LIN {X 0,Y 305.411,Z 367.044,A -85,B 0,C 180,E1 -16061.862,E2 -16061.862} C_VEL
LIN {X 0,Y 305.412,Z 367.294,A -85,B 0,C 180,E1 -16065.224,E2 -16065.224} C_VEL
LIN {X 0,Y 309.317,Z 377.708,A -85,B 0,C 180,E1 -16068.083,E2 -16068.083} C_VEL
LIN {X 0,Y 313.501,Z 390,A -85,B 0,C 180,E1 -16071.119,E2 -16071.119} C_VEL
LIN {X 0,Y 315.442,Z 396.314,A -85,B 0,C 180,E1 -16072.486,E2 -16072.486} C_VEL
LIN {X 0,Y 323.182,Z 411.941,A -85,B 0,C 180,E1 -16073.957,E2 -16073.957} C_VEL
LIN {X 0,Y 328.092,Z 423.496,A -85,B 0,C 180,E1 -16074.88,E2 -16074.88} C_VEL
LIN {X 0,Y 331.537,Z 444.039,A -85,B 0,C 180,E1 -16075.825,E2 -16075.825} C_VEL
LIN {X 0,Y 328.819,Z 524.988,A -85,B 0,C 180,E1 -16077.585,E2 -16077.585} C_VEL
LIN {X 0,Y 327.29,Z 565.254,A -85,B 0,C 180,E1 -16078.483,E2 -16078.483} C_VEL
LIN {X 0,Y 326.153,Z 580.481,A -85,B 0,C 180,E1 -16079.038,E2 -16079.038} C_VEL
LIN {X 0,Y 324.598,Z 594.646,A -85,B 0,C 180,E1 -16079.775,E2 -16079.775} C_VEL
LIN {X 0,Y 322.707,Z 608.869,A -85,B 0,C 180,E1 -16080.766,E2 -16080.766} C_VEL
LIN {X 0,Y 320.772,Z 621.593,A -85,B 0,C 180,E1 -16081.897,E2 -16081.897} C_VEL
LIN {X 0,Y 318.404,Z 634.299,A -85,B 0,C 180,E1 -16083.273,E2 -16083.273} C_VEL
LIN {X 0,Y 315.823,Z 647.117,A -85,B 0,C 180,E1 -16084.988,E2 -16084.988} C_VEL
LIN {X 0,Y 313.322,Z 658.678,A -85,B 0,C 180,E1 -16086.876,E2 -16086.876} C_VEL
LIN {X 0,Y 311.244,Z 668.516,A -85,B 0,C 180,E1 -16088.821,E2 -16088.821} C_VEL
LIN {X 0,Y 309.016,Z 678.081,A -85,B 0,C 180,E1 -16091.089,E2 -16091.089} C_VEL
LIN {X 0,Y 307.253,Z 686.052,A -85,B 0,C 180,E1 -16093.386,E2 -16093.386} C_VEL
LIN {X 0,Y 305.786,Z 693.474,A -85,B 0,C 180,E1 -16096.035,E2 -16096.035} C_VEL
LIN {X 0,Y 304.663,Z 699.365,A -85,B 0,C 180,E1 -16098.692,E2 -16098.692} C_VEL
LIN {X 0,Y 304.167,Z 702.846,A -85,B 0,C 180,E1 -16100.692,E2 -16100.692} C_VEL
LIN {X 0,Y 303.722,Z 706.396,A -85,B 0,C 180,E1 -16103.356,E2 -16103.356} C_VEL
LIN {X 0,Y 303.569,Z 708.739,A -85,B 0,C 180,E1 -16106.017,E2 -16106.017} C_VEL
LIN {X 0,Y 303.524,Z 709.928,A -85,B 0,C 180,E1 -16108.673,E2 -16108.673} C_VEL
LIN {X 0,Y 303.524,Z 709.94,A -85,B 0,C 180,E1 -16111.327,E2 -16111.327} C_VEL
LIN {X 0,Y 303.573,Z 708.8,A -85,B 0,C 180,E1 -16113.982,E2 -16113.982} C_VEL
LIN {X 0,Y 303.725,Z 706.51,A -85,B 0,C 180,E1 -16116.644,E2 -16116.644} C_VEL
LIN {X 0,Y 304.16,Z 703.02,A -85,B 0,C 180,E1 -16119.308,E2 -16119.308} C_VEL
LIN {X 0,Y 304.837,Z 698.241,A -85,B 0,C 180,E1 -16121.975,E2 -16121.975} C_VEL
LIN {X 0,Y 306.042,Z 692.044,A -85,B 0,C 180,E1 -16124.632,E2 -16124.632} C_VEL
LIN {X 0,Y 307.409,Z 685.357,A -85,B 0,C 180,E1 -16126.947,E2 -16126.947} C_VEL
LIN {X 0,Y 309.208,Z 677.258,A -85,B 0,C 180,E1 -16129.243,E2 -16129.243} C_VEL
LIN {X 0,Y 311.526,Z 667.524,A -85,B 0,C 180,E1 -16131.506,E2 -16131.506} C_VEL
LIN {X 0,Y 313.768,Z 656.8,A -85,B 0,C 180,E1 -16133.576,E2 -16133.576} C_VEL
LIN {X 0,Y 316.463,Z 644.635,A -85,B 0,C 180,E1 -16135.485,E2 -16135.485} C_VEL
LIN {X 0,Y 319.039,Z 631.238,A -85,B 0,C 180,E1 -16137.2,E2 -16137.2} C_VEL
LIN {X 0,Y 319.416,Z 629.216,A -85,B 0,C 180,E1 -16137.422,E2 -16137.422} C_VEL
LIN {X 0,Y 319.706,Z 624.316,A -85,B 0,C 180,E1 -16138.005,E2 -16138.005} C_VEL
LIN {X 0,Y 318.605,Z 616.252,A -85,B 0,C 180,E1 -16139.03,E2 -16139.03} C_VEL
LIN {X 0,Y 317.409,Z 607.963,A -85,B 0,C 180,E1 -16139.981,E2 -16139.981} C_VEL
LIN {X 0,Y 317.523,Z 602.64,A -85,B 0,C 180,E1 -16140.441,E2 -16140.441} C_VEL
LIN {X 0,Y 319.252,Z 588.464,A -85,B 0,C 180,E1 -16141.338,E2 -16141.338} C_VEL
LIN {X 0,Y 320.747,Z 573.705,A -85,B 0,C 180,E1 -16142.004,E2 -16142.004} C_VEL
LIN {X 0,Y 321.69,Z 558.805,A -85,B 0,C 180,E1 -16142.454,E2 -16142.454} C_VEL
LIN {X 0,Y 325.778,Z 445.6,A -85,B 0,C 180,E1 -16144.938,E2 -16144.938} C_VEL
LIN {X 0,Y 322.373,Z 425.482,A -85,B 0,C 180,E1 -16145.9,E2 -16145.9} C_VEL
LIN {X 0,Y 315.354,Z 409.904,A -85,B 0,C 180,E1 -16147.259,E2 -16147.259} C_VEL
LIN {X 0,Y 308.177,Z 395.852,A -85,B 0,C 180,E1 -16148.71,E2 -16148.71} C_VEL
LIN {X 0,Y 304.501,Z 384.759,A -85,B 0,C 180,E1 -16151.401,E2 -16151.401} C_VEL
LIN {X 0,Y 300.748,Z 374.308,A -85,B 0,C 180,E1 -16154.188,E2 -16154.188} C_VEL
LIN {X 0,Y 298.408,Z 368.151,A -85,B 0,C 180,E1 -16155.992,E2 -16155.992} C_VEL
LIN {X 0,Y 298.348,Z 367.948,A -85,B 0,C 180,E1 -16158.921,E2 -16158.921} C_VEL
LIN {X 0,Y 298.386,Z 367.941,A -85,B 0,C 180,E1 -16162.237,E2 -16162.237} C_VEL
LIN {X 0,Y 298.407,Z 367.933,A -85,B 0,C 180,E1 -16165.581,E2 -16165.581} C_VEL
LIN {X 0,Y 298.376,Z 367.928,A -85,B 0,C 180,E1 -16168.789,E2 -16168.789} C_VEL
LIN {X 0,Y 298.413,Z 367.926,A -85,B 0,C 180,E1 -16171.899,E2 -16171.899} C_VEL
LIN {X 0,Y 298.439,Z 367.934,A -85,B 0,C 180,E1 -16174.92,E2 -16174.92} C_VEL
LIN {X 0,Y 298.401,Z 367.92,A -85,B 0,C 180,E1 -16177.862,E2 -16177.862} C_VEL
LIN {X 0,Y 298.503,Z 367.927,A -85,B 0,C 180,E1 -16180.754,E2 -16180.754} C_VEL
LIN {X 0,Y 298.586,Z 367.911,A -85,B 0,C 180,E1 -16184.994,E2 -16184.994} C_VEL
LIN {X 0,Y 298.583,Z 367.892,A -85,B 0,C 180,E1 -16189.146,E2 -16189.146} C_VEL
LIN {X 0,Y 298.719,Z 367.902,A -85,B 0,C 180,E1 -16191.885,E2 -16191.885} C_VEL
LIN {X 0,Y 298.648,Z 367.885,A -85,B 0,C 180,E1 -16194.599,E2 -16194.599} C_VEL
LIN {X 0,Y 298.92,Z 367.875,A -85,B 0,C 180,E1 -16198.653,E2 -16198.653} C_VEL
LIN {X 0,Y 298.921,Z 367.849,A -85,B 0,C 180,E1 -16201.347,E2 -16201.347} C_VEL
LIN {X 0,Y 298.641,Z 367.905,A -85,B 0,C 180,E1 -16205.401,E2 -16205.401} C_VEL
LIN {X 0,Y 298.702,Z 367.875,A -85,B 0,C 180,E1 -16208.115,E2 -16208.115} C_VEL
LIN {X 0,Y 298.551,Z 367.909,A -85,B 0,C 180,E1 -16212.231,E2 -16212.231} C_VEL
LIN {X 0,Y 298.55,Z 367.905,A -85,B 0,C 180,E1 -16215.169,E2 -16215.169} C_VEL
LIN {X 0,Y 298.504,Z 367.905,A -85,B 0,C 180,E1 -16219.245,E2 -16219.245} C_VEL
LIN {X 0,Y 298.458,Z 367.924,A -85,B 0,C 180,E1 -16223.597,E2 -16223.597} C_VEL
LIN {X 0,Y 298.489,Z 367.924,A -85,B 0,C 180,E1 -16226.574,E2 -16226.574} C_VEL
LIN {X 0,Y 298.42,Z 367.92,A -85,B 0,C 180,E1 -16229.641,E2 -16229.641} C_VEL
LIN {X 0,Y 298.395,Z 367.939,A -85,B 0,C 180,E1 -16232.8,E2 -16232.8} C_VEL
LIN {X 0,Y 298.444,Z 367.935,A -85,B 0,C 180,E1 -16236.807,E2 -16236.807} C_VEL
LIN {X 0,Y 298.386,Z 367.89,A -85,B 0,C 180,E1 -16241.088,E2 -16241.088} C_VEL
LIN {X 0,Y 298.398,Z 367.931,A -85,B 0,C 180,E1 -16243.103,E2 -16243.103} C_VEL
LIN {X 0,Y 298.432,Z 368.054,A -85,B 0,C 180,E1 -16247.297,E2 -16247.297} C_VEL
LIN {X 0,Y 298.626,Z 368.899,A -85,B 0,C 180,E1 -16247.593,E2 -16247.593} C_VEL
LIN {X 0,Y 302.505,Z 376.069,A -85,B 0,C 180,E1 -16249.032,E2 -16249.032} C_VEL
LIN {X 0,Y 308.412,Z 392.412,A -85,B 0,C 180,E1 -16251.566,E2 -16251.566} C_VEL
LIN {X 0,Y 316.344,Z 409.427,A -85,B 0,C 180,E1 -16253.177,E2 -16253.177} C_VEL
LIN {X 0,Y 322.801,Z 424.458,A -85,B 0,C 180,E1 -16254.439,E2 -16254.439} C_VEL
LIN {X 0,Y 325.22,Z 441.813,A -85,B 0,C 180,E1 -16255.203,E2 -16255.203} C_VEL
LIN {X 0,Y 320.9,Z 562.756,A -85,B 0,C 180,E1 -16257.874,E2 -16257.874} C_VEL
LIN {X 0,Y 319.802,Z 578.013,A -85,B 0,C 180,E1 -16258.4,E2 -16258.4} C_VEL
LIN {X 0,Y 318.3,Z 592.161,A -85,B 0,C 180,E1 -16259.113,E2 -16259.113} C_VEL
LIN {X 0,Y 316.442,Z 606.126,A -85,B 0,C 180,E1 -16260.06,E2 -16260.06} C_VEL
LIN {X 0,Y 314.307,Z 619.886,A -85,B 0,C 180,E1 -16261.266,E2 -16261.266} C_VEL
LIN {X 0,Y 311.853,Z 632.809,A -85,B 0,C 180,E1 -16262.666,E2 -16262.666} C_VEL
LIN {X 0,Y 309.452,Z 644.715,A -85,B 0,C 180,E1 -16264.256,E2 -16264.256} C_VEL
LIN {X 0,Y 307.017,Z 655.77,A -85,B 0,C 180,E1 -16266.037,E2 -16266.037} C_VEL
LIN {X 0,Y 304.805,Z 665.842,A -85,B 0,C 180,E1 -16267.995,E2 -16267.995} C_VEL
LIN {X 0,Y 302.413,Z 675.711,A -85,B 0,C 180,E1 -16270.307,E2 -16270.307} C_VEL
LIN {X 0,Y 300.504,Z 683.894,A -85,B 0,C 180,E1 -16272.651,E2 -16272.651} C_VEL
LIN {X 0,Y 299.073,Z 690.659,A -85,B 0,C 180,E1 -16275.02,E2 -16275.02} C_VEL
LIN {X 0,Y 297.826,Z 696.924,A -85,B 0,C 180,E1 -16277.738,E2 -16277.738} C_VEL
LIN {X 0,Y 297.095,Z 701.755,A -85,B 0,C 180,E1 -16280.469,E2 -16280.469} C_VEL
LIN {X 0,Y 296.647,Z 705.286,A -85,B 0,C 180,E1 -16283.197,E2 -16283.197} C_VEL
LIN {X 0,Y 296.482,Z 707.609,A -85,B 0,C 180,E1 -16285.922,E2 -16285.922} C_VEL
LIN {X 0,Y 296.458,Z 708.776,A -85,B 0,C 180,E1 -16288.642,E2 -16288.642} C_VEL
LIN {X 0,Y 296.458,Z 708.774,A -85,B 0,C 180,E1 -16291.359,E2 -16291.359} C_VEL
LIN {X 0,Y 296.483,Z 707.601,A -85,B 0,C 180,E1 -16294.078,E2 -16294.078} C_VEL
LIN {X 0,Y 296.647,Z 705.268,A -85,B 0,C 180,E1 -16296.803,E2 -16296.803} C_VEL
LIN {X 0,Y 297.095,Z 701.72,A -85,B 0,C 180,E1 -16299.532,E2 -16299.532} C_VEL
LIN {X 0,Y 297.834,Z 696.875,A -85,B 0,C 180,E1 -16302.262,E2 -16302.262} C_VEL
LIN {X 0,Y 299.073,Z 690.605,A -85,B 0,C 180,E1 -16304.981,E2 -16304.981} C_VEL
LIN {X 0,Y 300.794,Z 682.716,A -85,B 0,C 180,E1 -16307.683,E2 -16307.683} C_VEL
LIN {X 0,Y 302.715,Z 674.287,A -85,B 0,C 180,E1 -16310.026,E2 -16310.026} C_VEL
LIN {X 0,Y 308.167,Z 654.094,A -85,B 0,C 180,E1 -16314.596,E2 -16314.596} C_VEL
LIN {X 0,Y 311.872,Z 642.327,A -85,B 0,C 180,E1 -16316.789,E2 -16316.789} C_VEL
LIN {X 0,Y 315.458,Z 630.417,A -85,B 0,C 180,E1 -16318.62,E2 -16318.62} C_VEL
LIN {X 0,Y 319.129,Z 617.583,A -85,B 0,C 180,E1 -16320.25,E2 -16320.25} C_VEL
LIN {X 0,Y 322.798,Z 603.816,A -85,B 0,C 180,E1 -16321.678,E2 -16321.678} C_VEL
LIN {X 0,Y 326.682,Z 587.895,A -85,B 0,C 180,E1 -16322.987,E2 -16322.987} C_VEL
LIN {X 0,Y 330.115,Z 572.099,A -85,B 0,C 180,E1 -16323.977,E2 -16323.977} C_VEL
LIN {X 0,Y 332.855,Z 556.74,A -85,B 0,C 180,E1 -16324.71,E2 -16324.71} C_VEL
LIN {X 0,Y 342.563,Z 489.987,A -85,B 0,C 180,E1 -16327.245,E2 -16327.245} C_VEL
LIN {X 0,Y 348.996,Z 451.001,A -85,B 0,C 180,E1 -16328.721,E2 -16328.721} C_VEL
LIN {X 0,Y 347.231,Z 446.356,A -85,B 0,C 180,E1 -16330.058,E2 -16330.058} C_VEL
LIN {X 0,Y 345.905,Z 443.202,A -85,B 0,C 180,E1 -16331.257,E2 -16331.257} C_VEL
LIN {X 0,Y 344.191,Z 439.714,A -85,B 0,C 180,E1 -16333.319,E2 -16333.319} C_VEL
LIN {X 0,Y 343.35,Z 438.48,A -85,B 0,C 180,E1 -16335.002,E2 -16335.002} C_VEL
LIN {X 0,Y 343.223,Z 438.552,A -85,B 0,C 180,E1 -16337.49,E2 -16337.49} C_VEL
LIN {X 0,Y 343.926,Z 439.872,A -85,B 0,C 180,E1 -16339.267,E2 -16339.267} C_VEL
LIN {X 0,Y 345.698,Z 444.259,A -85,B 0,C 180,E1 -16341.637,E2 -16341.637} C_VEL
LIN {X 0,Y 347.324,Z 448.856,A -85,B 0,C 180,E1 -16343.179,E2 -16343.179} C_VEL
LIN {X 0,Y 348.467,Z 452.55,A -85,B 0,C 180,E1 -16344.127,E2 -16344.127} C_VEL
LIN {X 0,Y 348.241,Z 454.474,A -85,B 0,C 180,E1 -16344.255,E2 -16344.255} C_VEL
LIN {X 0,Y 334.114,Z 539.694,A -85,B 0,C 180,E1 -16347.718,E2 -16347.718} C_VEL
LIN {X 0,Y 331.471,Z 555.843,A -85,B 0,C 180,E1 -16348.469,E2 -16348.469} C_VEL
LIN {X 0,Y 328.38,Z 571.369,A -85,B 0,C 180,E1 -16349.45,E2 -16349.45} C_VEL
LIN {X 0,Y 324.96,Z 586.557,A -85,B 0,C 180,E1 -16350.704,E2 -16350.704} C_VEL
LIN {X 0,Y 321.371,Z 600.391,A -85,B 0,C 180,E1 -16352.132,E2 -16352.132} C_VEL
LIN {X 0,Y 317.77,Z 613.05,A -85,B 0,C 180,E1 -16353.747,E2 -16353.747} C_VEL
LIN {X 0,Y 314.257,Z 624.641,A -85,B 0,C 180,E1 -16355.561,E2 -16355.561} C_VEL
LIN {X 0,Y 311.147,Z 634.413,A -85,B 0,C 180,E1 -16357.419,E2 -16357.419} C_VEL
LIN {X 0,Y 307.886,Z 644.112,A -85,B 0,C 180,E1 -16359.659,E2 -16359.659} C_VEL
LIN {X 0,Y 305.091,Z 651.899,A -85,B 0,C 180,E1 -16361.882,E2 -16361.882} C_VEL
LIN {X 0,Y 302.424,Z 659.117,A -85,B 0,C 180,E1 -16364.5,E2 -16364.5} C_VEL
LIN {X 0,Y 300.431,Z 664.653,A -85,B 0,C 180,E1 -16367.16,E2 -16367.16} C_VEL
LIN {X 0,Y 299.358,Z 667.8,A -85,B 0,C 180,E1 -16369.175,E2 -16369.175} C_VEL
LIN {X 0,Y 298.079,Z 670.711,A -85,B 0,C 180,E1 -16371.867,E2 -16371.867} C_VEL
LIN {X 0,Y 297.263,Z 672.207,A -85,B 0,C 180,E1 -16374.574,E2 -16374.574} C_VEL
LIN {X 0,Y 296.912,Z 672.286,A -85,B 0,C 180,E1 -16377.287,E2 -16377.287} C_VEL
LIN {X 0,Y 296.668,Z 670.948,A -85,B 0,C 180,E1 -16380,E2 -16380} C_VEL
LIN {X 0,Y 296.698,Z 668.154,A -85,B 0,C 180,E1 -16382.716,E2 -16382.716} C_VEL
LIN {X 0,Y 296.784,Z 665.05,A -85,B 0,C 180,E1 -16384.754,E2 -16384.754} C_VEL
LIN {X 0,Y 297.063,Z 660.107,A -85,B 0,C 180,E1 -16387.199,E2 -16387.199} C_VEL
LIN {X 0,Y 297.439,Z 654.084,A -85,B 0,C 180,E1 -16389.521,E2 -16389.521} C_VEL
LIN {X 0,Y 298.097,Z 646.353,A -85,B 0,C 180,E1 -16391.905,E2 -16391.905} C_VEL
LIN {X 0,Y 299.015,Z 638.312,A -85,B 0,C 180,E1 -16393.941,E2 -16393.941} C_VEL
LIN {X 0,Y 299.934,Z 628.773,A -85,B 0,C 180,E1 -16395.956,E2 -16395.956} C_VEL
LIN {X 0,Y 301.307,Z 617.06,A -85,B 0,C 180,E1 -16398.003,E2 -16398.003} C_VEL
LIN {X 0,Y 302.519,Z 605.387,A -85,B 0,C 180,E1 -16399.686,E2 -16399.686} C_VEL
LIN {X 0,Y 303.938,Z 592.777,A -85,B 0,C 180,E1 -16401.18,E2 -16401.18} C_VEL
LIN {X 0,Y 305.32,Z 579.078,A -85,B 0,C 180,E1 -16402.5,E2 -16402.5} C_VEL
LIN {X 0,Y 306.468,Z 564.482,A -85,B 0,C 180,E1 -16403.618,E2 -16403.618} C_VEL
LIN {X 0,Y 307.548,Z 548.938,A -85,B 0,C 180,E1 -16404.513,E2 -16404.513} C_VEL
LIN {X 0,Y 308.473,Z 531.327,A -85,B 0,C 180,E1 -16405.199,E2 -16405.199} C_VEL
LIN {X 0,Y 313.035,Z 438.431,A -85,B 0,C 180,E1 -16408.326,E2 -16408.326} C_VEL
LIN {X 0,Y 308.171,Z 405.676,A -85,B 0,C 180,E1 -16409.875,E2 -16409.875} C_VEL
LIN {X 0,Y 305.512,Z 398.037,A -85,B 0,C 180,E1 -16410.404,E2 -16410.404} C_VEL
LIN {X 0,Y 302.475,Z 384.617,A -85,B 0,C 180,E1 -16413.893,E2 -16413.893} C_VEL
LIN {X 0,Y 299.638,Z 372.911,A -85,B 0,C 180,E1 -16417.111,E2 -16417.111} C_VEL
LIN {X 0,Y 298.443,Z 368.214,A -85,B 0,C 180,E1 -16418.494,E2 -16418.494} C_VEL
LIN {X 0,Y 298.375,Z 367.944,A -85,B 0,C 180,E1 -16419.492,E2 -16419.492} C_VEL
LIN {X 0,Y 298.371,Z 367.944,A -85,B 0,C 180,E1 -16423.781,E2 -16423.781} C_VEL
LIN {X 0,Y 298.435,Z 368.42,A -85,B 0,C 180,E1 -16424.239,E2 -16424.239} C_VEL
LIN {X 0,Y 302.771,Z 379.718,A -85,B 0,C 180,E1 -16427.427,E2 -16427.427} C_VEL
LIN {X 0,Y 307.254,Z 392.856,A -85,B 0,C 180,E1 -16430.733,E2 -16430.733} C_VEL
LIN {X 0,Y 308.293,Z 396.188,A -85,B 0,C 180,E1 -16431.459,E2 -16431.459} C_VEL
LIN {X 0,Y 316.348,Z 411.985,A -85,B 0,C 180,E1 -16433.056,E2 -16433.056} C_VEL
LIN {X 0,Y 322.396,Z 425.621,A -85,B 0,C 180,E1 -16434.225,E2 -16434.225} C_VEL
LIN {X 0,Y 325.662,Z 445.137,A -85,B 0,C 180,E1 -16435.152,E2 -16435.152} C_VEL
LIN {X 0,Y 322.86,Z 525.012,A -85,B 0,C 180,E1 -16436.914,E2 -16436.914} C_VEL
LIN {X 0,Y 321.263,Z 565.177,A -85,B 0,C 180,E1 -16437.822,E2 -16437.822} C_VEL
LIN {X 0,Y 320.096,Z 580.432,A -85,B 0,C 180,E1 -16438.385,E2 -16438.385} C_VEL
LIN {X 0,Y 318.479,Z 594.609,A -85,B 0,C 180,E1 -16439.131,E2 -16439.131} C_VEL
LIN {X 0,Y 316.442,Z 609.431,A -85,B 0,C 180,E1 -16440.185,E2 -16440.185} C_VEL
LIN {X 0,Y 314.24,Z 623.112,A -85,B 0,C 180,E1 -16441.441,E2 -16441.441} C_VEL
LIN {X 0,Y 311.789,Z 635.543,A -85,B 0,C 180,E1 -16442.841,E2 -16442.841} C_VEL
LIN {X 0,Y 309.137,Z 648.15,A -85,B 0,C 180,E1 -16444.589,E2 -16444.589} C_VEL
LIN {X 0,Y 306.584,Z 659.378,A -85,B 0,C 180,E1 -16446.483,E2 -16446.483} C_VEL
LIN {X 0,Y 304.59,Z 668.5,A -85,B 0,C 180,E1 -16448.335,E2 -16448.335} C_VEL
LIN {X 0,Y 302.248,Z 678.066,A -85,B 0,C 180,E1 -16450.649,E2 -16450.649} C_VEL
LIN {X 0,Y 300.369,Z 686.037,A -85,B 0,C 180,E1 -16452.994,E2 -16452.994} C_VEL
LIN {X 0,Y 298.835,Z 693.46,A -85,B 0,C 180,E1 -16455.703,E2 -16455.703} C_VEL
LIN {X 0,Y 297.64,Z 699.351,A -85,B 0,C 180,E1 -16458.422,E2 -16458.422} C_VEL
LIN {X 0,Y 297.108,Z 702.832,A -85,B 0,C 180,E1 -16460.469,E2 -16460.469} C_VEL
LIN {X 0,Y 296.646,Z 706.383,A -85,B 0,C 180,E1 -16463.197,E2 -16463.197} C_VEL
LIN {X 0,Y 296.471,Z 708.725,A -85,B 0,C 180,E1 -16465.922,E2 -16465.922} C_VEL
LIN {X 0,Y 296.446,Z 709.914,A -85,B 0,C 180,E1 -16468.641,E2 -16468.641} C_VEL
LIN {X 0,Y 296.446,Z 709.926,A -85,B 0,C 180,E1 -16471.358,E2 -16471.358} C_VEL
LIN {X 0,Y 296.476,Z 708.786,A -85,B 0,C 180,E1 -16474.078,E2 -16474.078} C_VEL
LIN {X 0,Y 296.649,Z 706.495,A -85,B 0,C 180,E1 -16476.803,E2 -16476.803} C_VEL
LIN {X 0,Y 297.099,Z 703.005,A -85,B 0,C 180,E1 -16479.531,E2 -16479.531} C_VEL
LIN {X 0,Y 297.856,Z 698.225,A -85,B 0,C 180,E1 -16482.26,E2 -16482.26} C_VEL
LIN {X 0,Y 299.134,Z 692.027,A -85,B 0,C 180,E1 -16484.977,E2 -16484.977} C_VEL
LIN {X 0,Y 300.823,Z 684.238,A -85,B 0,C 180,E1 -16487.681,E2 -16487.681} C_VEL
LIN {X 0,Y 302.774,Z 675.935,A -85,B 0,C 180,E1 -16490.022,E2 -16490.022} C_VEL
LIN {X 0,Y 304.887,Z 667.503,A -85,B 0,C 180,E1 -16491.998,E2 -16491.998} C_VEL
LIN {X 0,Y 307.061,Z 657.467,A -85,B 0,C 180,E1 -16493.982,E2 -16493.982} C_VEL
LIN {X 0,Y 309.793,Z 645.673,A -85,B 0,C 180,E1 -16495.894,E2 -16495.894} C_VEL
LIN {X 0,Y 312.457,Z 632.555,A -85,B 0,C 180,E1 -16497.64,E2 -16497.64} C_VEL
LIN {X 0,Y 314.911,Z 619.45,A -85,B 0,C 180,E1 -16499.039,E2 -16499.039} C_VEL
LIN {X 0,Y 317.19,Z 605.239,A -85,B 0,C 180,E1 -16500.251,E2 -16500.251} C_VEL
LIN {X 0,Y 317.523,Z 602.64,A -85,B 0,C 180,E1 -16500.441,E2 -16500.441} C_VEL
LIN {X 0,Y 317.631,Z 597.225,A -85,B 0,C 180,E1 -16500.883,E2 -16500.883} C_VEL
LIN {X 0,Y 314.9,Z 581.34,A -85,B 0,C 180,E1 -16502.278,E2 -16502.278} C_VEL
LIN {X 0,Y 314.61,Z 575.744,A -85,B 0,C 180,E1 -16502.607,E2 -16502.607} C_VEL
LIN {X 0,Y 314.731,Z 573.829,A -85,B 0,C 180,E1 -16502.682,E2 -16502.682} C_VEL
LIN {X 0,Y 315.719,Z 558.663,A -85,B 0,C 180,E1 -16503.145,E2 -16503.145} C_VEL
LIN {X 0,Y 319.949,Z 446.756,A -85,B 0,C 180,E1 -16505.635,E2 -16505.635} C_VEL
LIN {X 0,Y 316.814,Z 428.216,A -85,B 0,C 180,E1 -16506.551,E2 -16506.551} C_VEL
LIN {X 0,Y 309.707,Z 412.421,A -85,B 0,C 180,E1 -16507.981,E2 -16507.981} C_VEL
LIN {X 0,Y 302.9,Z 399.352,A -85,B 0,C 180,E1 -16509.379,E2 -16509.379} C_VEL
LIN {X 0,Y 300.951,Z 395.526,A -85,B 0,C 180,E1 -16509.851,E2 -16509.851} C_VEL
LIN {X 0,Y 296.548,Z 382.513,A -85,B 0,C 180,E1 -16513.205,E2 -16513.205} C_VEL
LIN {X 0,Y 292.629,Z 372.347,A -85,B 0,C 180,E1 -16516.096,E2 -16516.096} C_VEL
LIN {X 0,Y 291.343,Z 368.975,A -85,B 0,C 180,E1 -16517.189,E2 -16517.189} C_VEL
LIN {X 0,Y 291.332,Z 368.811,A -85,B 0,C 180,E1 -16521.155,E2 -16521.155} C_VEL
LIN {X 0,Y 291.354,Z 368.805,A -85,B 0,C 180,E1 -16524.625,E2 -16524.625} C_VEL
LIN {X 0,Y 291.366,Z 368.802,A -85,B 0,C 180,E1 -16527.95,E2 -16527.95} C_VEL
LIN {X 0,Y 291.345,Z 368.816,A -85,B 0,C 180,E1 -16531.154,E2 -16531.154} C_VEL
LIN {X 0,Y 291.359,Z 368.809,A -85,B 0,C 180,E1 -16534.266,E2 -16534.266} C_VEL
LIN {X 0,Y 291.364,Z 368.797,A -85,B 0,C 180,E1 -16537.298,E2 -16537.298} C_VEL
LIN {X 0,Y 291.44,Z 368.807,A -85,B 0,C 180,E1 -16540.269,E2 -16540.269} C_VEL
LIN {X 0,Y 291.498,Z 368.788,A -85,B 0,C 180,E1 -16544.665,E2 -16544.665} C_VEL
LIN {X 0,Y 291.529,Z 368.77,A -85,B 0,C 180,E1 -16548.88,E2 -16548.88} C_VEL
LIN {X 0,Y 291.668,Z 368.778,A -85,B 0,C 180,E1 -16551.687,E2 -16551.687} C_VEL
LIN {X 0,Y 291.619,Z 368.761,A -85,B 0,C 180,E1 -16554.468,E2 -16554.468} C_VEL
LIN {X 0,Y 291.886,Z 368.751,A -85,B 0,C 180,E1 -16558.62,E2 -16558.62} C_VEL
LIN {X 0,Y 291.887,Z 368.724,A -85,B 0,C 180,E1 -16561.38,E2 -16561.38} C_VEL
LIN {X 0,Y 291.61,Z 368.78,A -85,B 0,C 180,E1 -16565.532,E2 -16565.532} C_VEL
LIN {X 0,Y 291.669,Z 368.757,A -85,B 0,C 180,E1 -16568.912,E2 -16568.912} C_VEL
LIN {X 0,Y 291.517,Z 368.779,A -85,B 0,C 180,E1 -16572.531,E2 -16572.531} C_VEL
LIN {X 0,Y 291.507,Z 368.784,A -85,B 0,C 180,E1 -16575.379,E2 -16575.379} C_VEL
LIN {X 0,Y 291.423,Z 368.786,A -85,B 0,C 180,E1 -16579.86,E2 -16579.86} C_VEL
LIN {X 0,Y 291.4,Z 368.795,A -85,B 0,C 180,E1 -16584.205,E2 -16584.205} C_VEL
LIN {X 0,Y 291.423,Z 368.81,A -85,B 0,C 180,E1 -16587.271,E2 -16587.271} C_VEL
LIN {X 0,Y 291.337,Z 368.803,A -85,B 0,C 180,E1 -16590.437,E2 -16590.437} C_VEL
LIN {X 0,Y 291.344,Z 368.806,A -85,B 0,C 180,E1 -16593.698,E2 -16593.698} C_VEL
LIN {X 0,Y 291.372,Z 368.807,A -85,B 0,C 180,E1 -16597.253,E2 -16597.253} C_VEL
LIN {X 0,Y 291.331,Z 368.764,A -85,B 0,C 180,E1 -16600.643,E2 -16600.643} C_VEL
LIN {X 0,Y 291.29,Z 368.812,A -85,B 0,C 180,E1 -16604.402,E2 -16604.402} C_VEL
LIN {X 0,Y 291.322,Z 368.967,A -85,B 0,C 180,E1 -16606.031,E2 -16606.031} C_VEL
LIN {X 0,Y 291.657,Z 370.251,A -85,B 0,C 180,E1 -16606.428,E2 -16606.428} C_VEL
LIN {X 0,Y 293.268,Z 372.793,A -85,B 0,C 180,E1 -16607.028,E2 -16607.028} C_VEL
LIN {X 0,Y 297.706,Z 381.398,A -85,B 0,C 180,E1 -16608.748,E2 -16608.748} C_VEL
LIN {X 0,Y 301.647,Z 392.41,A -85,B 0,C 180,E1 -16610.533,E2 -16610.533} C_VEL
LIN {X 0,Y 309.608,Z 409.51,A -85,B 0,C 180,E1 -16612.235,E2 -16612.235} C_VEL
LIN {X 0,Y 317.224,Z 426.908,A -85,B 0,C 180,E1 -16613.778,E2 -16613.778} C_VEL
LIN {X 0,Y 319.398,Z 443.039,A -85,B 0,C 180,E1 -16614.502,E2 -16614.502} C_VEL
LIN {X 0,Y 314.925,Z 562.876,A -85,B 0,C 180,E1 -16617.189,E2 -16617.189} C_VEL
LIN {X 0,Y 313.788,Z 578.087,A -85,B 0,C 180,E1 -16617.722,E2 -16617.722} C_VEL
LIN {X 0,Y 312.221,Z 592.215,A -85,B 0,C 180,E1 -16618.443,E2 -16618.443} C_VEL
LIN {X 0,Y 310.35,Z 605.809,A -85,B 0,C 180,E1 -16619.375,E2 -16619.375} C_VEL
LIN {X 0,Y 308.1,Z 619.92,A -85,B 0,C 180,E1 -16620.631,E2 -16620.631} C_VEL
LIN {X 0,Y 305.551,Z 632.838,A -85,B 0,C 180,E1 -16622.054,E2 -16622.054} C_VEL
LIN {X 0,Y 303.046,Z 644.741,A -85,B 0,C 180,E1 -16623.671,E2 -16623.671} C_VEL
LIN {X 0,Y 300.5,Z 655.742,A -85,B 0,C 180,E1 -16625.473,E2 -16625.473} C_VEL
LIN {X 0,Y 298.187,Z 665.863,A -85,B 0,C 180,E1 -16627.481,E2 -16627.481} C_VEL
LIN {X 0,Y 295.7,Z 675.73,A -85,B 0,C 180,E1 -16629.841,E2 -16629.841} C_VEL
LIN {X 0,Y 293.67,Z 683.912,A -85,B 0,C 180,E1 -16632.234,E2 -16632.234} C_VEL
LIN {X 0,Y 292.175,Z 690.676,A -85,B 0,C 180,E1 -16634.657,E2 -16634.657} C_VEL
LIN {X 0,Y 290.858,Z 696.94,A -85,B 0,C 180,E1 -16637.44,E2 -16637.44} C_VEL
LIN {X 0,Y 290.058,Z 701.771,A -85,B 0,C 180,E1 -16640.235,E2 -16640.235} C_VEL
LIN {X 0,Y 289.572,Z 705.301,A -85,B 0,C 180,E1 -16643.03,E2 -16643.03} C_VEL
LIN {X 0,Y 289.388,Z 707.623,A -85,B 0,C 180,E1 -16645.822,E2 -16645.822} C_VEL
LIN {X 0,Y 289.381,Z 708.79,A -85,B 0,C 180,E1 -16648.609,E2 -16648.609} C_VEL
LIN {X 0,Y 289.381,Z 708.788,A -85,B 0,C 180,E1 -16651.392,E2 -16651.392} C_VEL
LIN {X 0,Y 289.389,Z 707.614,A -85,B 0,C 180,E1 -16654.178,E2 -16654.178} C_VEL
LIN {X 0,Y 289.573,Z 705.282,A -85,B 0,C 180,E1 -16656.97,E2 -16656.97} C_VEL
LIN {X 0,Y 290.058,Z 701.734,A -85,B 0,C 180,E1 -16659.765,E2 -16659.765} C_VEL
LIN {X 0,Y 290.867,Z 696.889,A -85,B 0,C 180,E1 -16662.56,E2 -16662.56} C_VEL
LIN {X 0,Y 292.174,Z 690.619,A -85,B 0,C 180,E1 -16665.343,E2 -16665.343} C_VEL
LIN {X 0,Y 293.97,Z 682.731,A -85,B 0,C 180,E1 -16668.107,E2 -16668.107} C_VEL
LIN {X 0,Y 295.972,Z 674.303,A -85,B 0,C 180,E1 -16670.503,E2 -16670.503} C_VEL
LIN {X 0,Y 298.632,Z 664.994,A -85,B 0,C 180,E1 -16672.85,E2 -16672.85} C_VEL
LIN {X 0,Y 301.835,Z 655.393,A -85,B 0,C 180,E1 -16675.147,E2 -16675.147} C_VEL
LIN {X 0,Y 305.718,Z 644.038,A -85,B 0,C 180,E1 -16677.373,E2 -16677.373} C_VEL
LIN {X 0,Y 309.147,Z 633.635,A -85,B 0,C 180,E1 -16679.074,E2 -16679.074} C_VEL
LIN {X 0,Y 313.308,Z 620.392,A -85,B 0,C 180,E1 -16680.872,E2 -16680.872} C_VEL
LIN {X 0,Y 317.523,Z 605.973,A -85,B 0,C 180,E1 -16682.462,E2 -16682.462} C_VEL
LIN {X 0,Y 321.37,Z 591.772,A -85,B 0,C 180,E1 -16683.706,E2 -16683.706} C_VEL
LIN {X 0,Y 325.059,Z 576.525,A -85,B 0,C 180,E1 -16684.743,E2 -16684.743} C_VEL
LIN {X 0,Y 328.185,Z 561.072,A -85,B 0,C 180,E1 -16685.56,E2 -16685.56} C_VEL
LIN {X 0,Y 342.587,Z 472.807,A -85,B 0,C 180,E1 -16688.971,E2 -16688.971} C_VEL
LIN {X 0,Y 345.708,Z 455.092,A -85,B 0,C 180,E1 -16689.677,E2 -16689.677} C_VEL
LIN {X 0,Y 344.22,Z 451.001,A -85,B 0,C 180,E1 -16691.029,E2 -16691.029} C_VEL
LIN {X 0,Y 343.323,Z 448.898,A -85,B 0,C 180,E1 -16691.984,E2 -16691.984} C_VEL
LIN {X 0,Y 342.27,Z 446.478,A -85,B 0,C 180,E1 -16693.482,E2 -16693.482} C_VEL
LIN {X 0,Y 341.552,Z 445.346,A -85,B 0,C 180,E1 -16695.018,E2 -16695.018} C_VEL
LIN {X 0,Y 341.343,Z 445.359,A -85,B 0,C 180,E1 -16697.2,E2 -16697.2} C_VEL
LIN {X 0,Y 341.968,Z 446.519,A -85,B 0,C 180,E1 -16699.023,E2 -16699.023} C_VEL
LIN {X 0,Y 343.429,Z 450.717,A -85,B 0,C 180,E1 -16701.309,E2 -16701.309} C_VEL
LIN {X 0,Y 344.734,Z 454.921,A -85,B 0,C 180,E1 -16702.731,E2 -16702.731} C_VEL
LIN {X 0,Y 345.279,Z 456.712,A -85,B 0,C 180,E1 -16703.236,E2 -16703.236} C_VEL
LIN {X 0,Y 330.5,Z 539.876,A -85,B 0,C 180,E1 -16706.663,E2 -16706.663} C_VEL
LIN {X 0,Y 327.477,Z 556.799,A -85,B 0,C 180,E1 -16707.462,E2 -16707.462} C_VEL
LIN {X 0,Y 324.137,Z 572.305,A -85,B 0,C 180,E1 -16708.461,E2 -16708.461} C_VEL
LIN {X 0,Y 320.519,Z 587.161,A -85,B 0,C 180,E1 -16709.714,E2 -16709.714} C_VEL
LIN {X 0,Y 316.703,Z 600.792,A -85,B 0,C 180,E1 -16711.141,E2 -16711.141} C_VEL
LIN {X 0,Y 313.22,Z 612.264,A -85,B 0,C 180,E1 -16712.614,E2 -16712.614} C_VEL
LIN {X 0,Y 309.974,Z 622.171,A -85,B 0,C 180,E1 -16714.122,E2 -16714.122} C_VEL
LIN {X 0,Y 306.526,Z 632.284,A -85,B 0,C 180,E1 -16715.985,E2 -16715.985} C_VEL
LIN {X 0,Y 302.958,Z 642.188,A -85,B 0,C 180,E1 -16718.213,E2 -16718.213} C_VEL
LIN {X 0,Y 299.668,Z 650.461,A -85,B 0,C 180,E1 -16720.476,E2 -16720.476} C_VEL
LIN {X 0,Y 297.043,Z 657.196,A -85,B 0,C 180,E1 -16722.798,E2 -16722.798} C_VEL
LIN {X 0,Y 295.19,Z 661.928,A -85,B 0,C 180,E1 -16724.818,E2 -16724.818} C_VEL
LIN {X 0,Y 293.595,Z 665.761,A -85,B 0,C 180,E1 -16726.856,E2 -16726.856} C_VEL
LIN {X 0,Y 292.45,Z 668.698,A -85,B 0,C 180,E1 -16728.916,E2 -16728.916} C_VEL
LIN {X 0,Y 291.088,Z 671.413,A -85,B 0,C 180,E1 -16731.671,E2 -16731.671} C_VEL
LIN {X 0,Y 290.228,Z 672.722,A -85,B 0,C 180,E1 -16734.442,E2 -16734.442} C_VEL
LIN {X 0,Y 289.83,Z 672.625,A -85,B 0,C 180,E1 -16737.22,E2 -16737.22} C_VEL
LIN {X 0,Y 289.579,Z 671.115,A -85,B 0,C 180,E1 -16740,E2 -16740} C_VEL
LIN {X 0,Y 289.623,Z 668.153,A -85,B 0,C 180,E1 -16742.782,E2 -16742.782} C_VEL
LIN {X 0,Y 289.69,Z 664.88,A -85,B 0,C 180,E1 -16744.871,E2 -16744.871} C_VEL
LIN {X 0,Y 289.98,Z 660.108,A -85,B 0,C 180,E1 -16747.225,E2 -16747.225} C_VEL
LIN {X 0,Y 290.407,Z 653.553,A -85,B 0,C 180,E1 -16749.753,E2 -16749.753} C_VEL
LIN {X 0,Y 290.993,Z 646.844,A -85,B 0,C 180,E1 -16751.847,E2 -16751.847} C_VEL
LIN {X 0,Y 292.02,Z 637.336,A -85,B 0,C 180,E1 -16754.282,E2 -16754.282} C_VEL
LIN {X 0,Y 293.067,Z 627.187,A -85,B 0,C 180,E1 -16756.415,E2 -16756.415} C_VEL
LIN {X 0,Y 294.449,Z 615.458,A -85,B 0,C 180,E1 -16758.437,E2 -16758.437} C_VEL
LIN {X 0,Y 295.868,Z 602.078,A -85,B 0,C 180,E1 -16760.329,E2 -16760.329} C_VEL
LIN {X 0,Y 297.416,Z 588.811,A -85,B 0,C 180,E1 -16761.85,E2 -16761.85} C_VEL
LIN {X 0,Y 298.716,Z 575.078,A -85,B 0,C 180,E1 -16763.117,E2 -16763.117} C_VEL
LIN {X 0,Y 299.904,Z 559.878,A -85,B 0,C 180,E1 -16764.21,E2 -16764.21} C_VEL
LIN {X 0,Y 300.951,Z 544.242,A -85,B 0,C 180,E1 -16765.041,E2 -16765.041} C_VEL
LIN {X 0,Y 306.305,Z 439.003,A -85,B 0,C 180,E1 -16768.747,E2 -16768.747} C_VEL
LIN {X 0,Y 301.676,Z 407.703,A -85,B 0,C 180,E1 -16770.271,E2 -16770.271} C_VEL
LIN {X 0,Y 298.299,Z 398.11,A -85,B 0,C 180,E1 -16770.934,E2 -16770.934} C_VEL
LIN {X 0,Y 295.194,Z 384.603,A -85,B 0,C 180,E1 -16774.536,E2 -16774.536} C_VEL
LIN {X 0,Y 292.272,Z 372.655,A -85,B 0,C 180,E1 -16777.915,E2 -16777.915} C_VEL
LIN {X 0,Y 291.351,Z 368.926,A -85,B 0,C 180,E1 -16779.079,E2 -16779.079} C_VEL
LIN {X 0,Y 291.352,Z 368.963,A -85,B 0,C 180,E1 -16782.939,E2 -16782.939} C_VEL
LIN {X 0,Y 295.879,Z 380.758,A -85,B 0,C 180,E1 -16786.462,E2 -16786.462} C_VEL
LIN {X 0,Y 300.017,Z 392.699,A -85,B 0,C 180,E1 -16789.58,E2 -16789.58} C_VEL
LIN {X 0,Y 301.152,Z 396.004,A -85,B 0,C 180,E1 -16790.365,E2 -16790.365} C_VEL
LIN {X 0,Y 309.802,Z 412.692,A -85,B 0,C 180,E1 -16792.164,E2 -16792.164} C_VEL
LIN {X 0,Y 316.866,Z 428.449,A -85,B 0,C 180,E1 -16793.582,E2 -16793.582} C_VEL
LIN {X 0,Y 319.865,Z 446.903,A -85,B 0,C 180,E1 -16794.477,E2 -16794.477} C_VEL
LIN {X 0,Y 315.537,Z 560.976,A -85,B 0,C 180,E1 -16797.023,E2 -16797.023} C_VEL
LIN {X 0,Y 314.447,Z 576.05,A -85,B 0,C 180,E1 -16797.513,E2 -16797.513} C_VEL
LIN {X 0,Y 312.879,Z 590.817,A -85,B 0,C 180,E1 -16798.233,E2 -16798.233} C_VEL
LIN {X 0,Y 311.066,Z 604.645,A -85,B 0,C 180,E1 -16799.154,E2 -16799.154} C_VEL
LIN {X 0,Y 308.88,Z 618.424,A -85,B 0,C 180,E1 -16800.338,E2 -16800.338} C_VEL
LIN {X 0,Y 306.316,Z 631.689,A -85,B 0,C 180,E1 -16801.757,E2 -16801.757} C_VEL
LIN {X 0,Y 303.467,Z 644.976,A -85,B 0,C 180,E1 -16803.525,E2 -16803.525} C_VEL
LIN {X 0,Y 300.688,Z 656.759,A -85,B 0,C 180,E1 -16805.45,E2 -16805.45} C_VEL
LIN {X 0,Y 298.37,Z 667,A -85,B 0,C 180,E1 -16807.495,E2 -16807.495} C_VEL
LIN {X 0,Y 295.826,Z 676.823,A -85,B 0,C 180,E1 -16809.85,E2 -16809.85} C_VEL
LIN {X 0,Y 293.794,Z 684.977,A -85,B 0,C 180,E1 -16812.242,E2 -16812.242} C_VEL
LIN {X 0,Y 292.243,Z 691.728,A -85,B 0,C 180,E1 -16814.661,E2 -16814.661} C_VEL
LIN {X 0,Y 290.916,Z 697.98,A -85,B 0,C 180,E1 -16817.442,E2 -16817.442} C_VEL
LIN {X 0,Y 290.072,Z 702.819,A -85,B 0,C 180,E1 -16820.235,E2 -16820.235} C_VEL
LIN {X 0,Y 289.572,Z 706.369,A -85,B 0,C 180,E1 -16823.03,E2 -16823.03} C_VEL
LIN {X 0,Y 289.376,Z 708.712,A -85,B 0,C 180,E1 -16825.822,E2 -16825.822} C_VEL
LIN {X 0,Y 289.369,Z 709.901,A -85,B 0,C 180,E1 -16828.608,E2 -16828.608} C_VEL
LIN {X 0,Y 289.369,Z 709.913,A -85,B 0,C 180,E1 -16831.392,E2 -16831.392} C_VEL
LIN {X 0,Y 289.382,Z 708.772,A -85,B 0,C 180,E1 -16834.178,E2 -16834.178} C_VEL
LIN {X 0,Y 289.574,Z 706.481,A -85,B 0,C 180,E1 -16836.97,E2 -16836.97} C_VEL
LIN {X 0,Y 290.063,Z 702.99,A -85,B 0,C 180,E1 -16839.765,E2 -16839.765} C_VEL
LIN {X 0,Y 290.89,Z 698.209,A -85,B 0,C 180,E1 -16842.559,E2 -16842.559} C_VEL
LIN {X 0,Y 292.217,Z 692.01,A -85,B 0,C 180,E1 -16845.34,E2 -16845.34} C_VEL
LIN {X 0,Y 294.001,Z 684.219,A -85,B 0,C 180,E1 -16848.105,E2 -16848.105} C_VEL
LIN {X 0,Y 296.029,Z 675.915,A -85,B 0,C 180,E1 -16850.498,E2 -16850.498} C_VEL
LIN {X 0,Y 298.618,Z 665.905,A -85,B 0,C 180,E1 -16852.85,E2 -16852.85} C_VEL
LIN {X 0,Y 300.977,Z 655.681,A -85,B 0,C 180,E1 -16854.854,E2 -16854.854} C_VEL
LIN {X 0,Y 303.889,Z 643.435,A -85,B 0,C 180,E1 -16856.806,E2 -16856.806} C_VEL
LIN {X 0,Y 306.444,Z 631.174,A -85,B 0,C 180,E1 -16858.417,E2 -16858.417} C_VEL
LIN {X 0,Y 309.018,Z 617.775,A -85,B 0,C 180,E1 -16859.835,E2 -16859.835} C_VEL
LIN {X 0,Y 311.271,Z 603.736,A -85,B 0,C 180,E1 -16861.021,E2 -16861.021} C_VEL
LIN {X 0,Y 313.036,Z 589.852,A -85,B 0,C 180,E1 -16861.938,E2 -16861.938} C_VEL
LIN {X 0,Y 314.647,Z 574.678,A -85,B 0,C 180,E1 -16862.653,E2 -16862.653} C_VEL
LIN {X 0,Y 314.731,Z 573.829,A -85,B 0,C 180,E1 -16862.682,E2 -16862.682} C_VEL
LIN {X 0,Y 314.731,Z 568.088,A -85,B 0,C 180,E1 -16862.937,E2 -16862.937} C_VEL
LIN {X 0,Y 312.837,Z 558.826,A -85,B 0,C 180,E1 -16863.484,E2 -16863.484} C_VEL
LIN {X 0,Y 310.715,Z 549.529,A -85,B 0,C 180,E1 -16864.004,E2 -16864.004} C_VEL
LIN {X 0,Y 310.33,Z 543.724,A -85,B 0,C 180,E1 -16864.206,E2 -16864.206} C_VEL
LIN {X 0,Y 314.172,Z 447.853,A -85,B 0,C 180,E1 -16866.359,E2 -16866.359} C_VEL
LIN {X 0,Y 311.224,Z 430.675,A -85,B 0,C 180,E1 -16867.243,E2 -16867.243} C_VEL
LIN {X 0,Y 304.108,Z 415.064,A -85,B 0,C 180,E1 -16868.726,E2 -16868.726} C_VEL
LIN {X 0,Y 297.716,Z 402.734,A -85,B 0,C 180,E1 -16870.093,E2 -16870.093} C_VEL
LIN {X 0,Y 293.83,Z 395.597,A -85,B 0,C 180,E1 -16870.992,E2 -16870.992} C_VEL
LIN {X 0,Y 290.078,Z 384.698,A -85,B 0,C 180,E1 -16873.881,E2 -16873.881} C_VEL
LIN {X 0,Y 285.564,Z 373.039,A -85,B 0,C 180,E1 -16877.345,E2 -16877.345} C_VEL
LIN {X 0,Y 284.287,Z 369.886,A -85,B 0,C 180,E1 -16878.423,E2 -16878.423} C_VEL
LIN {X 0,Y 284.305,Z 369.695,A -85,B 0,C 180,E1 -16882.283,E2 -16882.283} C_VEL
LIN {X 0,Y 284.307,Z 369.686,A -85,B 0,C 180,E1 -16885.35,E2 -16885.35} C_VEL
LIN {X 0,Y 284.285,Z 369.683,A -85,B 0,C 180,E1 -16888.724,E2 -16888.724} C_VEL
LIN {X 0,Y 284.283,Z 369.684,A -85,B 0,C 180,E1 -16891.984,E2 -16891.984} C_VEL
LIN {X 0,Y 284.321,Z 369.688,A -85,B 0,C 180,E1 -16896.147,E2 -16896.147} C_VEL
LIN {X 0,Y 284.376,Z 369.684,A -85,B 0,C 180,E1 -16899.904,E2 -16899.904} C_VEL
LIN {X 0,Y 284.447,Z 369.662,A -85,B 0,C 180,E1 -16904.492,E2 -16904.492} C_VEL
LIN {X 0,Y 284.483,Z 369.649,A -85,B 0,C 180,E1 -16908.601,E2 -16908.601} C_VEL
LIN {X 0,Y 284.623,Z 369.653,A -85,B 0,C 180,E1 -16911.48,E2 -16911.48} C_VEL
LIN {X 0,Y 284.589,Z 369.637,A -85,B 0,C 180,E1 -16914.331,E2 -16914.331} C_VEL
LIN {X 0,Y 284.852,Z 369.628,A -85,B 0,C 180,E1 -16918.586,E2 -16918.586} C_VEL
LIN {X 0,Y 284.853,Z 369.599,A -85,B 0,C 180,E1 -16921.414,E2 -16921.414} C_VEL
LIN {X 0,Y 284.648,Z 369.627,A -85,B 0,C 180,E1 -16927.091,E2 -16927.091} C_VEL
LIN {X 0,Y 284.514,Z 369.662,A -85,B 0,C 180,E1 -16929.957,E2 -16929.957} C_VEL
LIN {X 0,Y 284.468,Z 369.649,A -85,B 0,C 180,E1 -16934.303,E2 -16934.303} C_VEL
LIN {X 0,Y 284.381,Z 369.666,A -85,B 0,C 180,E1 -16938.74,E2 -16938.74} C_VEL
LIN {X 0,Y 284.366,Z 369.682,A -85,B 0,C 180,E1 -16943.293,E2 -16943.293} C_VEL
LIN {X 0,Y 284.397,Z 369.684,A -85,B 0,C 180,E1 -16947.174,E2 -16947.174} C_VEL
LIN {X 0,Y 284.296,Z 369.688,A -85,B 0,C 180,E1 -16951.274,E2 -16951.274} C_VEL
LIN {X 0,Y 284.34,Z 369.68,A -85,B 0,C 180,E1 -16955.348,E2 -16955.348} C_VEL
LIN {X 0,Y 284.307,Z 369.66,A -85,B 0,C 180,E1 -16958.17,E2 -16958.17} C_VEL
LIN {X 0,Y 284.268,Z 369.661,A -85,B 0,C 180,E1 -16962.124,E2 -16962.124} C_VEL
LIN {X 0,Y 284.261,Z 369.888,A -85,B 0,C 180,E1 -16964.717,E2 -16964.717} C_VEL
LIN {X 0,Y 284.575,Z 371.106,A -85,B 0,C 180,E1 -16965.087,E2 -16965.087} C_VEL
LIN {X 0,Y 290.618,Z 381.832,A -85,B 0,C 180,E1 -16967.524,E2 -16967.524} C_VEL
LIN {X 0,Y 292.803,Z 386.627,A -85,B 0,C 180,E1 -16968.469,E2 -16968.469} C_VEL
LIN {X 0,Y 295.012,Z 392.642,A -85,B 0,C 180,E1 -16969.465,E2 -16969.465} C_VEL
LIN {X 0,Y 303.947,Z 411.631,A -85,B 0,C 180,E1 -16971.462,E2 -16971.462} C_VEL
LIN {X 0,Y 311.732,Z 429.747,A -85,B 0,C 180,E1 -16973.111,E2 -16973.111} C_VEL
LIN {X 0,Y 313.62,Z 444.341,A -85,B 0,C 180,E1 -16973.778,E2 -16973.778} C_VEL
LIN {X 0,Y 308.994,Z 562.992,A -85,B 0,C 180,E1 -16976.477,E2 -16976.477} C_VEL
LIN {X 0,Y 307.801,Z 578.159,A -85,B 0,C 180,E1 -16977.015,E2 -16977.015} C_VEL
LIN {X 0,Y 306.195,Z 592.268,A -85,B 0,C 180,E1 -16977.748,E2 -16977.748} C_VEL
LIN {X 0,Y 304.098,Z 606.821,A -85,B 0,C 180,E1 -16978.771,E2 -16978.771} C_VEL
LIN {X 0,Y 301.931,Z 619.955,A -85,B 0,C 180,E1 -16979.97,E2 -16979.97} C_VEL
LIN {X 0,Y 299.279,Z 632.868,A -85,B 0,C 180,E1 -16981.415,E2 -16981.415} C_VEL
LIN {X 0,Y 296.683,Z 644.767,A -85,B 0,C 180,E1 -16983.061,E2 -16983.061} C_VEL
LIN {X 0,Y 294.011,Z 655.765,A -85,B 0,C 180,E1 -16984.895,E2 -16984.895} C_VEL
LIN {X 0,Y 291.578,Z 665.925,A -85,B 0,C 180,E1 -16986.951,E2 -16986.951} C_VEL
LIN {X 0,Y 288.987,Z 675.75,A -85,B 0,C 180,E1 -16989.352,E2 -16989.352} C_VEL
LIN {X 0,Y 286.888,Z 683.93,A -85,B 0,C 180,E1 -16991.8,E2 -16991.8} C_VEL
LIN {X 0,Y 285.267,Z 690.693,A -85,B 0,C 180,E1 -16994.276,E2 -16994.276} C_VEL
LIN {X 0,Y 283.901,Z 696.956,A -85,B 0,C 180,E1 -16997.127,E2 -16997.127} C_VEL
LIN {X 0,Y 283.033,Z 701.786,A -85,B 0,C 180,E1 -16999.99,E2 -16999.99} C_VEL
LIN {X 0,Y 282.496,Z 705.316,A -85,B 0,C 180,E1 -17002.855,E2 -17002.855} C_VEL
LIN {X 0,Y 282.297,Z 707.637,A -85,B 0,C 180,E1 -17005.717,E2 -17005.717} C_VEL
LIN {X 0,Y 282.305,Z 708.803,A -85,B 0,C 180,E1 -17008.574,E2 -17008.574} C_VEL
LIN {X 0,Y 282.306,Z 708.801,A -85,B 0,C 180,E1 -17011.427,E2 -17011.427} C_VEL
LIN {X 0,Y 282.297,Z 707.628,A -85,B 0,C 180,E1 -17014.283,E2 -17014.283} C_VEL
LIN {X 0,Y 282.496,Z 705.295,A -85,B 0,C 180,E1 -17017.146,E2 -17017.146} C_VEL
LIN {X 0,Y 283.034,Z 701.748,A -85,B 0,C 180,E1 -17020.01,E2 -17020.01} C_VEL
LIN {X 0,Y 283.91,Z 696.903,A -85,B 0,C 180,E1 -17022.873,E2 -17022.873} C_VEL
LIN {X 0,Y 285.266,Z 690.633,A -85,B 0,C 180,E1 -17025.724,E2 -17025.724} C_VEL
LIN {X 0,Y 287.167,Z 682.746,A -85,B 0,C 180,E1 -17028.552,E2 -17028.552} C_VEL
LIN {X 0,Y 289.283,Z 674.34,A -85,B 0,C 180,E1 -17030.999,E2 -17030.999} C_VEL
LIN {X 0,Y 294.016,Z 660.943,A -85,B 0,C 180,E1 -17034.724,E2 -17034.724} C_VEL
LIN {X 0,Y 297.795,Z 650.769,A -85,B 0,C 180,E1 -17037.02,E2 -17037.02} C_VEL
LIN {X 0,Y 302.152,Z 638.765,A -85,B 0,C 180,E1 -17039.239,E2 -17039.239} C_VEL
LIN {X 0,Y 306.824,Z 625.53,A -85,B 0,C 180,E1 -17041.215,E2 -17041.215} C_VEL
LIN {X 0,Y 311.094,Z 612.345,A -85,B 0,C 180,E1 -17042.833,E2 -17042.833} C_VEL
LIN {X 0,Y 315.665,Z 597.264,A -85,B 0,C 180,E1 -17044.304,E2 -17044.304} C_VEL
LIN {X 0,Y 319.552,Z 582.981,A -85,B 0,C 180,E1 -17045.401,E2 -17045.401} C_VEL
LIN {X 0,Y 323.494,Z 566.161,A -85,B 0,C 180,E1 -17046.397,E2 -17046.397} C_VEL
LIN {X 0,Y 326.849,Z 548.508,A -85,B 0,C 180,E1 -17047.163,E2 -17047.163} C_VEL
LIN {X 0,Y 337.78,Z 485.154,A -85,B 0,C 180,E1 -17049.632,E2 -17049.632} C_VEL
LIN {X 0,Y 342.67,Z 459.418,A -85,B 0,C 180,E1 -17050.637,E2 -17050.637} C_VEL
LIN {X 0,Y 341.456,Z 455.993,A -85,B 0,C 180,E1 -17051.978,E2 -17051.978} C_VEL
LIN {X 0,Y 340.25,Z 453.072,A -85,B 0,C 180,E1 -17053.816,E2 -17053.816} C_VEL
LIN {X 0,Y 339.656,Z 452.163,A -85,B 0,C 180,E1 -17055.291,E2 -17055.291} C_VEL
LIN {X 0,Y 339.589,Z 452.329,A -85,B 0,C 180,E1 -17057.522,E2 -17057.522} C_VEL
LIN {X 0,Y 340.071,Z 453.494,A -85,B 0,C 180,E1 -17058.985,E2 -17058.985} C_VEL
LIN {X 0,Y 341.195,Z 457.148,A -85,B 0,C 180,E1 -17060.967,E2 -17060.967} C_VEL
LIN {X 0,Y 342.208,Z 460.954,A -85,B 0,C 180,E1 -17062.271,E2 -17062.271} C_VEL
LIN {X 0,Y 324.583,Z 554.028,A -85,B 0,C 180,E1 -17066.207,E2 -17066.207} C_VEL
LIN {X 0,Y 321.486,Z 568.053,A -85,B 0,C 180,E1 -17067.058,E2 -17067.058} C_VEL
LIN {X 0,Y 317.928,Z 582.064,A -85,B 0,C 180,E1 -17068.145,E2 -17068.145} C_VEL
LIN {X 0,Y 313.77,Z 596.416,A -85,B 0,C 180,E1 -17069.551,E2 -17069.551} C_VEL
LIN {X 0,Y 309.519,Z 609.61,A -85,B 0,C 180,E1 -17071.151,E2 -17071.151} C_VEL
LIN {X 0,Y 305.325,Z 621.688,A -85,B 0,C 180,E1 -17072.96,E2 -17072.96} C_VEL
LIN {X 0,Y 301.002,Z 633.373,A -85,B 0,C 180,E1 -17075.148,E2 -17075.148} C_VEL
LIN {X 0,Y 297.17,Z 643.112,A -85,B 0,C 180,E1 -17077.403,E2 -17077.403} C_VEL
LIN {X 0,Y 293.667,Z 651.232,A -85,B 0,C 180,E1 -17079.695,E2 -17079.695} C_VEL
LIN {X 0,Y 290.43,Z 658.738,A -85,B 0,C 180,E1 -17082.393,E2 -17082.393} C_VEL
LIN {X 0,Y 287.86,Z 664.548,A -85,B 0,C 180,E1 -17085.146,E2 -17085.146} C_VEL
LIN {X 0,Y 286.319,Z 667.86,A -85,B 0,C 180,E1 -17087.237,E2 -17087.237} C_VEL
LIN {X 0,Y 284.734,Z 671.056,A -85,B 0,C 180,E1 -17090.051,E2 -17090.051} C_VEL
LIN {X 0,Y 283.626,Z 672.858,A -85,B 0,C 180,E1 -17092.883,E2 -17092.883} C_VEL
LIN {X 0,Y 282.928,Z 673.277,A -85,B 0,C 180,E1 -17095.726,E2 -17095.726} C_VEL
LIN {X 0,Y 282.584,Z 672.29,A -85,B 0,C 180,E1 -17098.575,E2 -17098.575} C_VEL
LIN {X 0,Y 282.481,Z 669.861,A -85,B 0,C 180,E1 -17101.426,E2 -17101.426} C_VEL
LIN {X 0,Y 282.547,Z 667.036,A -85,B 0,C 180,E1 -17103.565,E2 -17103.565} C_VEL
LIN {X 0,Y 282.783,Z 661.918,A -85,B 0,C 180,E1 -17106.421,E2 -17106.421} C_VEL
LIN {X 0,Y 283.081,Z 656.893,A -85,B 0,C 180,E1 -17108.567,E2 -17108.567} C_VEL
LIN {X 0,Y 283.696,Z 649.671,A -85,B 0,C 180,E1 -17111.069,E2 -17111.069} C_VEL
LIN {X 0,Y 284.561,Z 640.723,A -85,B 0,C 180,E1 -17113.57,E2 -17113.57} C_VEL
LIN {X 0,Y 285.618,Z 631.411,A -85,B 0,C 180,E1 -17115.704,E2 -17115.704} C_VEL
LIN {X 0,Y 286.836,Z 620.196,A -85,B 0,C 180,E1 -17117.835,E2 -17117.835} C_VEL
LIN {X 0,Y 288.266,Z 607.814,A -85,B 0,C 180,E1 -17119.772,E2 -17119.772} C_VEL
LIN {X 0,Y 289.828,Z 594.15,A -85,B 0,C 180,E1 -17121.516,E2 -17121.516} C_VEL
LIN {X 0,Y 291.249,Z 580.831,A -85,B 0,C 180,E1 -17122.884,E2 -17122.884} C_VEL
LIN {X 0,Y 292.533,Z 565.893,A -85,B 0,C 180,E1 -17124.106,E2 -17124.106} C_VEL
LIN {X 0,Y 293.69,Z 550.046,A -85,B 0,C 180,E1 -17125.088,E2 -17125.088} C_VEL
LIN {X 0,Y 294.655,Z 533.236,A -85,B 0,C 180,E1 -17125.804,E2 -17125.804} C_VEL
LIN {X 0,Y 299.584,Z 439.968,A -85,B 0,C 180,E1 -17129.153,E2 -17129.153} C_VEL
LIN {X 0,Y 295.275,Z 410.189,A -85,B 0,C 180,E1 -17130.637,E2 -17130.637} C_VEL
LIN {X 0,Y 291.03,Z 398.175,A -85,B 0,C 180,E1 -17131.487,E2 -17131.487} C_VEL
LIN {X 0,Y 288.154,Z 385.38,A -85,B 0,C 180,E1 -17134.97,E2 -17134.97} C_VEL
LIN {X 0,Y 285.121,Z 373.217,A -85,B 0,C 180,E1 -17138.499,E2 -17138.499} C_VEL
LIN {X 0,Y 284.336,Z 369.807,A -85,B 0,C 180,E1 -17139.607,E2 -17139.607} C_VEL
LIN {X 0,Y 284.264,Z 369.808,A -85,B 0,C 180,E1 -17141.64,E2 -17141.64} C_VEL
LIN {X 0,Y 284.66,Z 371.346,A -85,B 0,C 180,E1 -17142.211,E2 -17142.211} C_VEL
LIN {X 0,Y 288.451,Z 380.499,A -85,B 0,C 180,E1 -17145.043,E2 -17145.043} C_VEL
LIN {X 0,Y 292.096,Z 390.449,A -85,B 0,C 180,E1 -17147.797,E2 -17147.797} C_VEL
LIN {X 0,Y 293.938,Z 395.876,A -85,B 0,C 180,E1 -17149.188,E2 -17149.188} C_VEL
LIN {X 0,Y 301.859,Z 410.578,A -85,B 0,C 180,E1 -17150.925,E2 -17150.925} C_VEL
LIN {X 0,Y 308.938,Z 425.598,A -85,B 0,C 180,E1 -17152.412,E2 -17152.412} C_VEL
LIN {X 0,Y 311.533,Z 431.778,A -85,B 0,C 180,E1 -17152.953,E2 -17152.953} C_VEL
LIN {X 0,Y 314.082,Z 447.923,A -85,B 0,C 180,E1 -17153.751,E2 -17153.751} C_VEL
LIN {X 0,Y 309.986,Z 552.444,A -85,B 0,C 180,E1 -17156.111,E2 -17156.111} C_VEL
LIN {X 0,Y 309.05,Z 569.823,A -85,B 0,C 180,E1 -17156.581,E2 -17156.581} C_VEL
LIN {X 0,Y 307.542,Z 585.068,A -85,B 0,C 180,E1 -17157.227,E2 -17157.227} C_VEL
LIN {X 0,Y 305.741,Z 599.275,A -85,B 0,C 180,E1 -17158.082,E2 -17158.082} C_VEL
LIN {X 0,Y 303.531,Z 613.432,A -85,B 0,C 180,E1 -17159.205,E2 -17159.205} C_VEL
LIN {X 0,Y 300.88,Z 627.482,A -85,B 0,C 180,E1 -17160.625,E2 -17160.625} C_VEL
LIN {X 0,Y 298.139,Z 640.376,A -85,B 0,C 180,E1 -17162.253,E2 -17162.253} C_VEL
LIN {X 0,Y 295.591,Z 651.213,A -85,B 0,C 180,E1 -17163.905,E2 -17163.905} C_VEL
LIN {X 0,Y 292.903,Z 662.171,A -85,B 0,C 180,E1 -17165.927,E2 -17165.927} C_VEL
LIN {X 0,Y 290.541,Z 671.398,A -85,B 0,C 180,E1 -17167.98,E2 -17167.98} C_VEL
LIN {X 0,Y 288.142,Z 680.469,A -85,B 0,C 180,E1 -17170.405,E2 -17170.405} C_VEL
LIN {X 0,Y 286.207,Z 688.001,A -85,B 0,C 180,E1 -17172.862,E2 -17172.862} C_VEL
LIN {X 0,Y 284.634,Z 695.027,A -85,B 0,C 180,E1 -17175.705,E2 -17175.705} C_VEL
LIN {X 0,Y 283.402,Z 700.553,A -85,B 0,C 180,E1 -17178.557,E2 -17178.557} C_VEL
LIN {X 0,Y 282.744,Z 704.736,A -85,B 0,C 180,E1 -17181.423,E2 -17181.423} C_VEL
LIN {X 0,Y 282.35,Z 707.959,A -85,B 0,C 180,E1 -17184.653,E2 -17184.653} C_VEL
LIN {X 0,Y 282.293,Z 709.435,A -85,B 0,C 180,E1 -17187.146,E2 -17187.146} C_VEL
LIN {X 0,Y 282.275,Z 710.043,A -85,B 0,C 180,E1 -17190,E2 -17190} C_VEL
LIN {X 0,Y 282.295,Z 709.47,A -85,B 0,C 180,E1 -17192.854,E2 -17192.854} C_VEL
LIN {X 0,Y 282.384,Z 707.758,A -85,B 0,C 180,E1 -17195.713,E2 -17195.713} C_VEL
LIN {X 0,Y 282.746,Z 704.875,A -85,B 0,C 180,E1 -17198.577,E2 -17198.577} C_VEL
LIN {X 0,Y 283.375,Z 700.752,A -85,B 0,C 180,E1 -17201.444,E2 -17201.444} C_VEL
LIN {X 0,Y 284.594,Z 695.28,A -85,B 0,C 180,E1 -17204.297,E2 -17204.297} C_VEL
LIN {X 0,Y 286.18,Z 688.31,A -85,B 0,C 180,E1 -17207.139,E2 -17207.139} C_VEL
LIN {X 0,Y 288.06,Z 680.848,A -85,B 0,C 180,E1 -17209.601,E2 -17209.601} C_VEL
LIN {X 0,Y 290.459,Z 671.859,A -85,B 0,C 180,E1 -17212.027,E2 -17212.027} C_VEL
LIN {X 0,Y 293.041,Z 661.599,A -85,B 0,C 180,E1 -17214.307,E2 -17214.307} C_VEL
LIN {X 0,Y 295.978,Z 649.825,A -85,B 0,C 180,E1 -17216.437,E2 -17216.437} C_VEL
LIN {X 0,Y 298.811,Z 637.563,A -85,B 0,C 180,E1 -17218.251,E2 -17218.251} C_VEL
LIN {X 0,Y 301.677,Z 624.019,A -85,B 0,C 180,E1 -17219.865,E2 -17219.865} C_VEL
LIN {X 0,Y 304.147,Z 609.995,A -85,B 0,C 180,E1 -17221.208,E2 -17221.208} C_VEL
LIN {X 0,Y 306.205,Z 596.093,A -85,B 0,C 180,E1 -17222.251,E2 -17222.251} C_VEL
LIN {X 0,Y 307.995,Z 581.622,A -85,B 0,C 180,E1 -17223.059,E2 -17223.059} C_VEL
LIN {X 0,Y 309.317,Z 567.036,A -85,B 0,C 180,E1 -17223.63,E2 -17223.63} C_VEL
LIN {X 0,Y 310.33,Z 543.724,A -85,B 0,C 180,E1 -17224.206,E2 -17224.206} C_VEL
LIN {X 0,Y 309.992,Z 537.92,A -85,B 0,C 180,E1 -17224.408,E2 -17224.408} C_VEL
LIN {X 0,Y 306.078,Z 519.262,A -85,B 0,C 180,E1 -17225.433,E2 -17225.433} C_VEL
LIN {X 0,Y 305.835,Z 513.456,A -85,B 0,C 180,E1 -17225.63,E2 -17225.63} C_VEL
LIN {X 0,Y 308.445,Z 448.978,A -85,B 0,C 180,E1 -17227.109,E2 -17227.109} C_VEL
LIN {X 0,Y 305.912,Z 433.852,A -85,B 0,C 180,E1 -17227.907,E2 -17227.907} C_VEL
LIN {X 0,Y 299.448,Z 419.505,A -85,B 0,C 180,E1 -17229.305,E2 -17229.305} C_VEL
LIN {X 0,Y 293.151,Z 407.15,A -85,B 0,C 180,E1 -17230.704,E2 -17230.704} C_VEL
LIN {X 0,Y 286.676,Z 395.541,A -85,B 0,C 180,E1 -17232.238,E2 -17232.238} C_VEL
LIN {X 0,Y 283.713,Z 387.011,A -85,B 0,C 180,E1 -17234.583,E2 -17234.583} C_VEL
LIN {X 0,Y 279.63,Z 376.689,A -85,B 0,C 180,E1 -17237.754,E2 -17237.754} C_VEL
LIN {X 0,Y 277.258,Z 370.797,A -85,B 0,C 180,E1 -17239.745,E2 -17239.745} C_VEL
LIN {X 0,Y 277.251,Z 370.577,A -85,B 0,C 180,E1 -17242.528,E2 -17242.528} C_VEL
LIN {X 0,Y 277.246,Z 370.575,A -85,B 0,C 180,E1 -17246.104,E2 -17246.104} C_VEL
LIN {X 0,Y 277.262,Z 370.563,A -85,B 0,C 180,E1 -17249.538,E2 -17249.538} C_VEL
LIN {X 0,Y 277.292,Z 370.55,A -85,B 0,C 180,E1 -17252.857,E2 -17252.857} C_VEL
LIN {X 0,Y 277.282,Z 370.565,A -85,B 0,C 180,E1 -17256.075,E2 -17256.075} C_VEL
LIN {X 0,Y 277.324,Z 370.566,A -85,B 0,C 180,E1 -17260.765,E2 -17260.765} C_VEL
LIN {X 0,Y 277.41,Z 370.55,A -85,B 0,C 180,E1 -17265.324,E2 -17265.324} C_VEL
LIN {X 0,Y 277.458,Z 370.524,A -85,B 0,C 180,E1 -17269.787,E2 -17269.787} C_VEL
LIN {X 0,Y 277.629,Z 370.526,A -85,B 0,C 180,E1 -17272.728,E2 -17272.728} C_VEL
LIN {X 0,Y 277.818,Z 370.504,A -85,B 0,C 180,E1 -17278.55,E2 -17278.55} C_VEL
LIN {X 0,Y 277.819,Z 370.475,A -85,B 0,C 180,E1 -17281.449,E2 -17281.449} C_VEL
LIN {X 0,Y 277.606,Z 370.502,A -85,B 0,C 180,E1 -17287.272,E2 -17287.272} C_VEL
LIN {X 0,Y 277.458,Z 370.545,A -85,B 0,C 180,E1 -17290.213,E2 -17290.213} C_VEL
LIN {X 0,Y 277.414,Z 370.529,A -85,B 0,C 180,E1 -17294.675,E2 -17294.675} C_VEL
LIN {X 0,Y 277.328,Z 370.541,A -85,B 0,C 180,E1 -17299.235,E2 -17299.235} C_VEL
LIN {X 0,Y 277.329,Z 370.55,A -85,B 0,C 180,E1 -17303.92,E2 -17303.92} C_VEL
LIN {X 0,Y 277.326,Z 370.568,A -85,B 0,C 180,E1 -17307.505,E2 -17307.505} C_VEL
LIN {X 0,Y 277.272,Z 370.555,A -85,B 0,C 180,E1 -17310.481,E2 -17310.481} C_VEL
LIN {X 0,Y 277.247,Z 370.56,A -85,B 0,C 180,E1 -17313.896,E2 -17313.896} C_VEL
LIN {X 0,Y 277.264,Z 370.553,A -85,B 0,C 180,E1 -17317.47,E2 -17317.47} C_VEL
LIN {X 0,Y 277.208,Z 370.525,A -85,B 0,C 180,E1 -17321.237,E2 -17321.237} C_VEL
LIN {X 0,Y 277.2,Z 370.658,A -85,B 0,C 180,E1 -17323.2,E2 -17323.2} C_VEL
LIN {X 0,Y 277.466,Z 371.711,A -85,B 0,C 180,E1 -17323.601,E2 -17323.601} C_VEL
LIN {X 0,Y 285.506,Z 386.251,A -85,B 0,C 180,E1 -17327.081,E2 -17327.081} C_VEL
LIN {X 0,Y 287.46,Z 390.494,A -85,B 0,C 180,E1 -17327.956,E2 -17327.956} C_VEL
LIN {X 0,Y 288.696,Z 393.352,A -85,B 0,C 180,E1 -17328.401,E2 -17328.401} C_VEL
LIN {X 0,Y 298.903,Z 415.136,A -85,B 0,C 180,E1 -17330.79,E2 -17330.79} C_VEL
LIN {X 0,Y 306.341,Z 432.841,A -85,B 0,C 180,E1 -17332.436,E2 -17332.436} C_VEL
LIN {X 0,Y 307.887,Z 445.733,A -85,B 0,C 180,E1 -17333.028,E2 -17333.028} C_VEL
LIN {X 0,Y 303.111,Z 563.11,A -85,B 0,C 180,E1 -17335.737,E2 -17335.737} C_VEL
LIN {X 0,Y 301.858,Z 578.233,A -85,B 0,C 180,E1 -17336.28,E2 -17336.28} C_VEL
LIN {X 0,Y 300.21,Z 592.321,A -85,B 0,C 180,E1 -17337.024,E2 -17337.024} C_VEL
LIN {X 0,Y 298.083,Z 606.661,A -85,B 0,C 180,E1 -17338.047,E2 -17338.047} C_VEL
LIN {X 0,Y 295.796,Z 619.989,A -85,B 0,C 180,E1 -17339.281,E2 -17339.281} C_VEL
LIN {X 0,Y 293.052,Z 632.897,A -85,B 0,C 180,E1 -17340.749,E2 -17340.749} C_VEL
LIN {X 0,Y 290.35,Z 644.792,A -85,B 0,C 180,E1 -17342.424,E2 -17342.424} C_VEL
LIN {X 0,Y 287.556,Z 655.787,A -85,B 0,C 180,E1 -17344.29,E2 -17344.29} C_VEL
LIN {X 0,Y 284.97,Z 666.083,A -85,B 0,C 180,E1 -17346.419,E2 -17346.419} C_VEL
LIN {X 0,Y 282.284,Z 675.769,A -85,B 0,C 180,E1 -17348.838,E2 -17348.838} C_VEL
LIN {X 0,Y 280.097,Z 683.948,A -85,B 0,C 180,E1 -17351.342,E2 -17351.342} C_VEL
LIN {X 0,Y 278.368,Z 690.71,A -85,B 0,C 180,E1 -17353.876,E2 -17353.876} C_VEL
LIN {X 0,Y 276.951,Z 696.972,A -85,B 0,C 180,E1 -17356.798,E2 -17356.798} C_VEL
LIN {X 0,Y 275.999,Z 701.801,A -85,B 0,C 180,E1 -17359.733,E2 -17359.733} C_VEL
LIN {X 0,Y 275.444,Z 705.33,A -85,B 0,C 180,E1 -17362.671,E2 -17362.671} C_VEL
LIN {X 0,Y 275.211,Z 707.651,A -85,B 0,C 180,E1 -17365.606,E2 -17365.606} C_VEL
LIN {X 0,Y 275.231,Z 708.817,A -85,B 0,C 180,E1 -17368.537,E2 -17368.537} C_VEL
LIN {X 0,Y 275.232,Z 708.815,A -85,B 0,C 180,E1 -17371.463,E2 -17371.463} C_VEL
LIN {X 0,Y 275.212,Z 707.641,A -85,B 0,C 180,E1 -17374.394,E2 -17374.394} C_VEL
LIN {X 0,Y 275.444,Z 705.309,A -85,B 0,C 180,E1 -17377.33,E2 -17377.33} C_VEL
LIN {X 0,Y 275.999,Z 701.761,A -85,B 0,C 180,E1 -17380.268,E2 -17380.268} C_VEL
LIN {X 0,Y 276.959,Z 696.917,A -85,B 0,C 180,E1 -17383.202,E2 -17383.202} C_VEL
LIN {X 0,Y 278.371,Z 690.648,A -85,B 0,C 180,E1 -17386.124,E2 -17386.124} C_VEL
LIN {X 0,Y 280.396,Z 682.761,A -85,B 0,C 180,E1 -17389.017,E2 -17389.017} C_VEL
LIN {X 0,Y 282.27,Z 675.686,A -85,B 0,C 180,E1 -17391.163,E2 -17391.163} C_VEL
LIN {X 0,Y 285.757,Z 667.124,A -85,B 0,C 180,E1 -17393.942,E2 -17393.942} C_VEL
LIN {X 0,Y 289.321,Z 658.224,A -85,B 0,C 180,E1 -17396.316,E2 -17396.316} C_VEL
LIN {X 0,Y 293.572,Z 647.748,A -85,B 0,C 180,E1 -17398.607,E2 -17398.607} C_VEL
LIN {X 0,Y 297.665,Z 637.284,A -85,B 0,C 180,E1 -17400.506,E2 -17400.506} C_VEL
LIN {X 0,Y 302.254,Z 625.132,A -85,B 0,C 180,E1 -17402.33,E2 -17402.33} C_VEL
LIN {X 0,Y 307.255,Z 610.877,A -85,B 0,C 180,E1 -17404.084,E2 -17404.084} C_VEL
LIN {X 0,Y 312.188,Z 595.563,A -85,B 0,C 180,E1 -17405.553,E2 -17405.553} C_VEL
LIN {X 0,Y 316.27,Z 581.444,A -85,B 0,C 180,E1 -17406.621,E2 -17406.621} C_VEL
LIN {X 0,Y 320.152,Z 565.969,A -85,B 0,C 180,E1 -17407.53,E2 -17407.53} C_VEL
LIN {X 0,Y 323.747,Z 548.438,A -85,B 0,C 180,E1 -17408.295,E2 -17408.295} C_VEL
LIN {X 0,Y 335.757,Z 484.082,A -85,B 0,C 180,E1 -17410.833,E2 -17410.833} C_VEL
LIN {X 0,Y 339.817,Z 464.162,A -85,B 0,C 180,E1 -17411.615,E2 -17411.615} C_VEL
LIN {X 0,Y 339.173,Z 462.103,A -85,B 0,C 180,E1 -17412.505,E2 -17412.505} C_VEL
LIN {X 0,Y 338.311,Z 459.775,A -85,B 0,C 180,E1 -17414.043,E2 -17414.043} C_VEL
LIN {X 0,Y 337.929,Z 459.094,A -85,B 0,C 180,E1 -17415,E2 -17415} C_VEL
LIN {X 0,Y 337.733,Z 459.144,A -85,B 0,C 180,E1 -17417.385,E2 -17417.385} C_VEL
LIN {X 0,Y 338.111,Z 460.202,A -85,B 0,C 180,E1 -17418.767,E2 -17418.767} C_VEL
LIN {X 0,Y 338.986,Z 463.579,A -85,B 0,C 180,E1 -17420.61,E2 -17420.61} C_VEL
LIN {X 0,Y 339.415,Z 465.303,A -85,B 0,C 180,E1 -17421.273,E2 -17421.273} C_VEL
LIN {X 0,Y 321.421,Z 554.341,A -85,B 0,C 180,E1 -17425.068,E2 -17425.068} C_VEL
LIN {X 0,Y 317.685,Z 570.06,A -85,B 0,C 180,E1 -17426.042,E2 -17426.042} C_VEL
LIN {X 0,Y 313.924,Z 583.543,A -85,B 0,C 180,E1 -17427.119,E2 -17427.119} C_VEL
LIN {X 0,Y 309.104,Z 598.782,A -85,B 0,C 180,E1 -17428.661,E2 -17428.661} C_VEL
LIN {X 0,Y 304.634,Z 611.515,A -85,B 0,C 180,E1 -17430.264,E2 -17430.264} C_VEL
LIN {X 0,Y 300.193,Z 623.215,A -85,B 0,C 180,E1 -17432.081,E2 -17432.081} C_VEL
LIN {X 0,Y 295.587,Z 634.604,A -85,B 0,C 180,E1 -17434.284,E2 -17434.284} C_VEL
LIN {X 0,Y 291.65,Z 643.766,A -85,B 0,C 180,E1 -17436.461,E2 -17436.461} C_VEL
LIN {X 0,Y 287.764,Z 652.102,A -85,B 0,C 180,E1 -17438.885,E2 -17438.885} C_VEL
LIN {X 0,Y 284.591,Z 658.64,A -85,B 0,C 180,E1 -17441.275,E2 -17441.275} C_VEL
LIN {X 0,Y 281.738,Z 664.542,A -85,B 0,C 180,E1 -17444.074,E2 -17444.074} C_VEL
LIN {X 0,Y 279.472,Z 668.932,A -85,B 0,C 180,E1 -17446.919,E2 -17446.919} C_VEL
LIN {X 0,Y 277.801,Z 671.883,A -85,B 0,C 180,E1 -17449.8,E2 -17449.8} C_VEL
LIN {X 0,Y 276.6,Z 673.46,A -85,B 0,C 180,E1 -17452.701,E2 -17452.701} C_VEL
LIN {X 0,Y 275.872,Z 673.657,A -85,B 0,C 180,E1 -17455.617,E2 -17455.617} C_VEL
LIN {X 0,Y 275.503,Z 672.455,A -85,B 0,C 180,E1 -17458.538,E2 -17458.538} C_VEL
LIN {X 0,Y 275.402,Z 669.827,A -85,B 0,C 180,E1 -17461.462,E2 -17461.462} C_VEL
LIN {X 0,Y 275.465,Z 666.899,A -85,B 0,C 180,E1 -17463.657,E2 -17463.657} C_VEL
LIN {X 0,Y 275.722,Z 661.53,A -85,B 0,C 180,E1 -17466.586,E2 -17466.586} C_VEL
LIN {X 0,Y 276.091,Z 655.375,A -85,B 0,C 180,E1 -17469.155,E2 -17469.155} C_VEL
LIN {X 0,Y 276.756,Z 647.668,A -85,B 0,C 180,E1 -17471.722,E2 -17471.722} C_VEL
LIN {X 0,Y 277.805,Z 638.19,A -85,B 0,C 180,E1 -17474.28,E2 -17474.28} C_VEL
LIN {X 0,Y 278.849,Z 627.946,A -85,B 0,C 180,E1 -17476.55,E2 -17476.55} C_VEL
LIN {X 0,Y 280.281,Z 616.407,A -85,B 0,C 180,E1 -17478.645,E2 -17478.645} C_VEL
LIN {X 0,Y 281.592,Z 604.416,A -85,B 0,C 180,E1 -17480.452,E2 -17480.452} C_VEL
LIN {X 0,Y 283.349,Z 589.95,A -85,B 0,C 180,E1 -17482.226,E2 -17482.226} C_VEL
LIN {X 0,Y 284.731,Z 576.408,A -85,B 0,C 180,E1 -17483.561,E2 -17483.561} C_VEL
LIN {X 0,Y 285.944,Z 561.764,A -85,B 0,C 180,E1 -17484.698,E2 -17484.698} C_VEL
LIN {X 0,Y 287.048,Z 545.946,A -85,B 0,C 180,E1 -17485.613,E2 -17485.613} C_VEL
LIN {X 0,Y 288.699,Z 515.284,A -85,B 0,C 180,E1 -17486.816,E2 -17486.816} C_VEL
LIN {X 0,Y 292.77,Z 440.439,A -85,B 0,C 180,E1 -17489.599,E2 -17489.599} C_VEL
LIN {X 0,Y 288.693,Z 412.104,A -85,B 0,C 180,E1 -17491.056,E2 -17491.056} C_VEL
LIN {X 0,Y 283.768,Z 398.111,A -85,B 0,C 180,E1 -17492.068,E2 -17492.068} C_VEL
LIN {X 0,Y 280.746,Z 384.695,A -85,B 0,C 180,E1 -17495.839,E2 -17495.839} C_VEL
LIN {X 0,Y 277.681,Z 372.311,A -85,B 0,C 180,E1 -17499.548,E2 -17499.548} C_VEL
LIN {X 0,Y 277.256,Z 370.694,A -85,B 0,C 180,E1 -17500.191,E2 -17500.191} C_VEL
LIN {X 0,Y 277.309,Z 371.062,A -85,B 0,C 180,E1 -17500.508,E2 -17500.508} C_VEL
LIN {X 0,Y 281.413,Z 381.221,A -85,B 0,C 180,E1 -17503.821,E2 -17503.821} C_VEL
LIN {X 0,Y 285.148,Z 390.927,A -85,B 0,C 180,E1 -17506.642,E2 -17506.642} C_VEL
LIN {X 0,Y 286.914,Z 396.068,A -85,B 0,C 180,E1 -17507.983,E2 -17507.983} C_VEL
LIN {X 0,Y 294.527,Z 409.738,A -85,B 0,C 180,E1 -17509.736,E2 -17509.736} C_VEL
LIN {X 0,Y 302.066,Z 425.177,A -85,B 0,C 180,E1 -17511.394,E2 -17511.394} C_VEL
LIN {X 0,Y 306.171,Z 434.865,A -85,B 0,C 180,E1 -17512.284,E2 -17512.284} C_VEL
LIN {X 0,Y 308.309,Z 448.654,A -85,B 0,C 180,E1 -17512.985,E2 -17512.985} C_VEL
LIN {X 0,Y 304.61,Z 539.853,A -85,B 0,C 180,E1 -17515.077,E2 -17515.077} C_VEL
LIN {X 0,Y 303.395,Z 566.32,A -85,B 0,C 180,E1 -17515.723,E2 -17515.723} C_VEL
LIN {X 0,Y 301.986,Z 582.019,A -85,B 0,C 180,E1 -17516.346,E2 -17516.346} C_VEL
LIN {X 0,Y 300.061,Z 597.004,A -85,B 0,C 180,E1 -17517.205,E2 -17517.205} C_VEL
LIN {X 0,Y 297.72,Z 611.835,A -85,B 0,C 180,E1 -17518.357,E2 -17518.357} C_VEL
LIN {X 0,Y 295.027,Z 626.064,A -85,B 0,C 180,E1 -17519.786,E2 -17519.786} C_VEL
LIN {X 0,Y 292.122,Z 639.204,A -85,B 0,C 180,E1 -17521.434,E2 -17521.434} C_VEL
LIN {X 0,Y 289.176,Z 651.195,A -85,B 0,C 180,E1 -17523.281,E2 -17523.281} C_VEL
LIN {X 0,Y 286.332,Z 662.154,A -85,B 0,C 180,E1 -17525.338,E2 -17525.338} C_VEL
LIN {X 0,Y 283.947,Z 671.383,A -85,B 0,C 180,E1 -17527.44,E2 -17527.44} C_VEL
LIN {X 0,Y 281.41,Z 680.454,A -85,B 0,C 180,E1 -17529.916,E2 -17529.916} C_VEL
LIN {X 0,Y 279.385,Z 687.987,A -85,B 0,C 180,E1 -17532.43,E2 -17532.43} C_VEL
LIN {X 0,Y 277.679,Z 695.013,A -85,B 0,C 180,E1 -17535.339,E2 -17535.339} C_VEL
LIN {X 0,Y 276.391,Z 700.54,A -85,B 0,C 180,E1 -17538.263,E2 -17538.263} C_VEL
LIN {X 0,Y 275.684,Z 704.722,A -85,B 0,C 180,E1 -17541.201,E2 -17541.201} C_VEL
LIN {X 0,Y 275.29,Z 707.66,A -85,B 0,C 180,E1 -17544.139,E2 -17544.139} C_VEL
LIN {X 0,Y 275.205,Z 709.421,A -85,B 0,C 180,E1 -17547.072,E2 -17547.072} C_VEL
LIN {X 0,Y 275.2,Z 710.03,A -85,B 0,C 180,E1 -17550,E2 -17550} C_VEL
LIN {X 0,Y 275.206,Z 709.456,A -85,B 0,C 180,E1 -17552.927,E2 -17552.927} C_VEL
LIN {X 0,Y 275.296,Z 707.743,A -85,B 0,C 180,E1 -17555.861,E2 -17555.861} C_VEL
LIN {X 0,Y 275.684,Z 704.86,A -85,B 0,C 180,E1 -17558.798,E2 -17558.798} C_VEL
LIN {X 0,Y 276.364,Z 700.736,A -85,B 0,C 180,E1 -17561.738,E2 -17561.738} C_VEL
LIN {X 0,Y 277.639,Z 695.263,A -85,B 0,C 180,E1 -17564.663,E2 -17564.663} C_VEL
LIN {X 0,Y 279.335,Z 688.292,A -85,B 0,C 180,E1 -17567.573,E2 -17567.573} C_VEL
LIN {X 0,Y 281.328,Z 680.829,A -85,B 0,C 180,E1 -17570.09,E2 -17570.09} C_VEL
LIN {X 0,Y 283.866,Z 671.838,A -85,B 0,C 180,E1 -17572.566,E2 -17572.566} C_VEL
LIN {X 0,Y 286.621,Z 661.143,A -85,B 0,C 180,E1 -17574.983,E2 -17574.983} C_VEL
LIN {X 0,Y 289.593,Z 649.799,A -85,B 0,C 180,E1 -17577.067,E2 -17577.067} C_VEL
LIN {X 0,Y 292.541,Z 637.533,A -85,B 0,C 180,E1 -17578.913,E2 -17578.913} C_VEL
LIN {X 0,Y 295.515,Z 623.984,A -85,B 0,C 180,E1 -17580.553,E2 -17580.553} C_VEL
LIN {X 0,Y 298.088,Z 609.898,A -85,B 0,C 180,E1 -17581.922,E2 -17581.922} C_VEL
LIN {X 0,Y 300.224,Z 596.041,A -85,B 0,C 180,E1 -17582.974,E2 -17582.974} C_VEL
LIN {X 0,Y 302.072,Z 581.55,A -85,B 0,C 180,E1 -17583.793,E2 -17583.793} C_VEL
LIN {X 0,Y 303.423,Z 566.926,A -85,B 0,C 180,E1 -17584.373,E2 -17584.373} C_VEL
LIN {X 0,Y 305.059,Z 530.573,A -85,B 0,C 180,E1 -17585.249,E2 -17585.249} C_VEL
LIN {X 0,Y 305.835,Z 513.456,A -85,B 0,C 180,E1 -17585.63,E2 -17585.63} C_VEL
LIN {X 0,Y 305.569,Z 507.656,A -85,B 0,C 180,E1 -17585.83,E2 -17585.83} C_VEL
LIN {X 0,Y 301.581,Z 489.073,A -85,B 0,C 180,E1 -17586.917,E2 -17586.917} C_VEL
LIN {X 0,Y 301.281,Z 483.273,A -85,B 0,C 180,E1 -17587.129,E2 -17587.129} C_VEL
LIN {X 0,Y 302.706,Z 449.472,A -85,B 0,C 180,E1 -17587.916,E2 -17587.916} C_VEL
LIN {X 0,Y 300.565,Z 436.822,A -85,B 0,C 180,E1 -17588.611,E2 -17588.611} C_VEL
LIN {X 0,Y 294.634,Z 423.541,A -85,B 0,C 180,E1 -17589.945,E2 -17589.945} C_VEL
LIN {X 0,Y 288.347,Z 411.084,A -85,B 0,C 180,E1 -17591.398,E2 -17591.398} C_VEL
LIN {X 0,Y 281.652,Z 399.222,A -85,B 0,C 180,E1 -17593.007,E2 -17593.007} C_VEL
LIN {X 0,Y 279.56,Z 395.352,A -85,B 0,C 180,E1 -17593.587,E2 -17593.587} C_VEL
LIN {X 0,Y 275.326,Z 384.159,A -85,B 0,C 180,E1 -17596.936,E2 -17596.936} C_VEL
LIN {X 0,Y 271.364,Z 374.536,A -85,B 0,C 180,E1 -17600.134,E2 -17600.134} C_VEL
LIN {X 0,Y 270.208,Z 371.652,A -85,B 0,C 180,E1 -17601.224,E2 -17601.224} C_VEL
LIN {X 0,Y 270.197,Z 371.441,A -85,B 0,C 180,E1 -17605.094,E2 -17605.094} C_VEL
LIN {X 0,Y 270.184,Z 371.44,A -85,B 0,C 180,E1 -17609.136,E2 -17609.136} C_VEL
LIN {X 0,Y 270.223,Z 371.433,A -85,B 0,C 180,E1 -17612.163,E2 -17612.163} C_VEL
LIN {X 0,Y 270.227,Z 371.45,A -85,B 0,C 180,E1 -17615.542,E2 -17615.542} C_VEL
LIN {X 0,Y 270.277,Z 371.444,A -85,B 0,C 180,E1 -17620.242,E2 -17620.242} C_VEL
LIN {X 0,Y 270.378,Z 371.42,A -85,B 0,C 180,E1 -17624.934,E2 -17624.934} C_VEL
LIN {X 0,Y 270.41,Z 371.4,A -85,B 0,C 180,E1 -17629.518,E2 -17629.518} C_VEL
LIN {X 0,Y 270.585,Z 371.404,A -85,B 0,C 180,E1 -17632.538,E2 -17632.538} C_VEL
LIN {X 0,Y 270.783,Z 371.38,A -85,B 0,C 180,E1 -17638.513,E2 -17638.513} C_VEL
LIN {X 0,Y 270.785,Z 371.35,A -85,B 0,C 180,E1 -17641.487,E2 -17641.487} C_VEL
LIN {X 0,Y 270.566,Z 371.377,A -85,B 0,C 180,E1 -17647.462,E2 -17647.462} C_VEL
LIN {X 0,Y 270.41,Z 371.423,A -85,B 0,C 180,E1 -17650.482,E2 -17650.482} C_VEL
LIN {X 0,Y 270.373,Z 371.41,A -85,B 0,C 180,E1 -17655.066,E2 -17655.066} C_VEL
LIN {X 0,Y 270.274,Z 371.418,A -85,B 0,C 180,E1 -17659.757,E2 -17659.757} C_VEL
LIN {X 0,Y 270.274,Z 371.423,A -85,B 0,C 180,E1 -17664.585,E2 -17664.585} C_VEL
LIN {X 0,Y 270.27,Z 371.445,A -85,B 0,C 180,E1 -17667.909,E2 -17667.909} C_VEL
LIN {X 0,Y 270.184,Z 371.446,A -85,B 0,C 180,E1 -17671.348,E2 -17671.348} C_VEL
LIN {X 0,Y 270.201,Z 371.437,A -85,B 0,C 180,E1 -17674.905,E2 -17674.905} C_VEL
LIN {X 0,Y 270.197,Z 371.404,A -85,B 0,C 180,E1 -17678.71,E2 -17678.71} C_VEL
LIN {X 0,Y 270.182,Z 371.523,A -85,B 0,C 180,E1 -17681.62,E2 -17681.62} C_VEL
LIN {X 0,Y 270.462,Z 372.714,A -85,B 0,C 180,E1 -17682.085,E2 -17682.085} C_VEL
LIN {X 0,Y 277.206,Z 384.688,A -85,B 0,C 180,E1 -17685.225,E2 -17685.225} C_VEL
LIN {X 0,Y 281.316,Z 392.439,A -85,B 0,C 180,E1 -17687.012,E2 -17687.012} C_VEL
LIN {X 0,Y 285.506,Z 400.411,A -85,B 0,C 180,E1 -17688.061,E2 -17688.061} C_VEL
LIN {X 0,Y 294.243,Z 419.57,A -85,B 0,C 180,E1 -17690.179,E2 -17690.179} C_VEL
LIN {X 0,Y 300.963,Z 435.58,A -85,B 0,C 180,E1 -17691.721,E2 -17691.721} C_VEL
LIN {X 0,Y 302.219,Z 446.991,A -85,B 0,C 180,E1 -17692.247,E2 -17692.247} C_VEL
LIN {X 0,Y 297.282,Z 563.231,A -85,B 0,C 180,E1 -17694.968,E2 -17694.968} C_VEL
LIN {X 0,Y 295.999,Z 578.308,A -85,B 0,C 180,E1 -17695.519,E2 -17695.519} C_VEL
LIN {X 0,Y 294.278,Z 592.375,A -85,B 0,C 180,E1 -17696.271,E2 -17696.271} C_VEL
LIN {X 0,Y 291.968,Z 607.314,A -85,B 0,C 180,E1 -17697.359,E2 -17697.359} C_VEL
LIN {X 0,Y 289.387,Z 621.59,A -85,B 0,C 180,E1 -17698.728,E2 -17698.728} C_VEL
LIN {X 0,Y 286.557,Z 634.207,A -85,B 0,C 180,E1 -17700.222,E2 -17700.222} C_VEL
LIN {X 0,Y 283.769,Z 645.878,A -85,B 0,C 180,E1 -17701.929,E2 -17701.929} C_VEL
LIN {X 0,Y 280.673,Z 657.579,A -85,B 0,C 180,E1 -17704.011,E2 -17704.011} C_VEL
LIN {X 0,Y 278.062,Z 667.413,A -85,B 0,C 180,E1 -17706.147,E2 -17706.147} C_VEL
LIN {X 0,Y 275.287,Z 677.016,A -85,B 0,C 180,E1 -17708.667,E2 -17708.667} C_VEL
LIN {X 0,Y 273.031,Z 685.003,A -85,B 0,C 180,E1 -17711.231,E2 -17711.231} C_VEL
LIN {X 0,Y 271.066,Z 692.441,A -85,B 0,C 180,E1 -17714.203,E2 -17714.203} C_VEL
LIN {X 0,Y 269.659,Z 698.337,A -85,B 0,C 180,E1 -17717.201,E2 -17717.201} C_VEL
LIN {X 0,Y 268.954,Z 701.816,A -85,B 0,C 180,E1 -17719.461,E2 -17719.461} C_VEL
LIN {X 0,Y 268.366,Z 705.345,A -85,B 0,C 180,E1 -17722.476,E2 -17722.476} C_VEL
LIN {X 0,Y 268.13,Z 707.666,A -85,B 0,C 180,E1 -17725.49,E2 -17725.49} C_VEL
LIN {X 0,Y 268.136,Z 708.831,A -85,B 0,C 180,E1 -17728.498,E2 -17728.498} C_VEL
LIN {X 0,Y 268.137,Z 708.829,A -85,B 0,C 180,E1 -17731.502,E2 -17731.502} C_VEL
LIN {X 0,Y 268.13,Z 707.655,A -85,B 0,C 180,E1 -17734.51,E2 -17734.51} C_VEL
LIN {X 0,Y 268.367,Z 705.322,A -85,B 0,C 180,E1 -17737.524,E2 -17737.524} C_VEL
LIN {X 0,Y 268.954,Z 701.775,A -85,B 0,C 180,E1 -17740.54,E2 -17740.54} C_VEL
LIN {X 0,Y 269.988,Z 696.931,A -85,B 0,C 180,E1 -17743.549,E2 -17743.549} C_VEL
LIN {X 0,Y 271.463,Z 690.662,A -85,B 0,C 180,E1 -17746.546,E2 -17746.546} C_VEL
LIN {X 0,Y 273.625,Z 682.779,A -85,B 0,C 180,E1 -17749.506,E2 -17749.506} C_VEL
LIN {X 0,Y 274.939,Z 678.283,A -85,B 0,C 180,E1 -17750.97,E2 -17750.97} C_VEL
LIN {X 0,Y 278.379,Z 670.468,A -85,B 0,C 180,E1 -17753.825,E2 -17753.825} C_VEL
LIN {X 0,Y 282.546,Z 661.05,A -85,B 0,C 180,E1 -17756.598,E2 -17756.598} C_VEL
LIN {X 0,Y 286.9,Z 651.25,A -85,B 0,C 180,E1 -17758.934,E2 -17758.934} C_VEL
LIN {X 0,Y 291.843,Z 639.724,A -85,B 0,C 180,E1 -17761.182,E2 -17761.182} C_VEL
LIN {X 0,Y 297.026,Z 627.147,A -85,B 0,C 180,E1 -17763.173,E2 -17763.173} C_VEL
LIN {X 0,Y 302.267,Z 613.484,A -85,B 0,C 180,E1 -17764.929,E2 -17764.929} C_VEL
LIN {X 0,Y 307.565,Z 598.544,A -85,B 0,C 180,E1 -17766.45,E2 -17766.45} C_VEL
LIN {X 0,Y 311.735,Z 585.546,A -85,B 0,C 180,E1 -17767.496,E2 -17767.496} C_VEL
LIN {X 0,Y 316.519,Z 568.45,A -85,B 0,C 180,E1 -17768.569,E2 -17768.569} C_VEL
LIN {X 0,Y 320.745,Z 549.79,A -85,B 0,C 180,E1 -17769.414,E2 -17769.414} C_VEL
LIN {X 0,Y 333.555,Z 485.838,A -85,B 0,C 180,E1 -17771.956,E2 -17771.956} C_VEL
LIN {X 0,Y 337.229,Z 468.99,A -85,B 0,C 180,E1 -17772.614,E2 -17772.614} C_VEL
LIN {X 0,Y 336.367,Z 466.44,A -85,B 0,C 180,E1 -17774.302,E2 -17774.302} C_VEL
LIN {X 0,Y 336.013,Z 465.905,A -85,B 0,C 180,E1 -17775.328,E2 -17775.328} C_VEL
LIN {X 0,Y 335.964,Z 466.197,A -85,B 0,C 180,E1 -17777.718,E2 -17777.718} C_VEL
LIN {X 0,Y 336.211,Z 467.107,A -85,B 0,C 180,E1 -17778.697,E2 -17778.697} C_VEL
LIN {X 0,Y 336.823,Z 470.046,A -85,B 0,C 180,E1 -17780.268,E2 -17780.268} C_VEL
LIN {X 0,Y 318.802,Z 554.019,A -85,B 0,C 180,E1 -17783.864,E2 -17783.864} C_VEL
LIN {X 0,Y 315.574,Z 566.811,A -85,B 0,C 180,E1 -17784.618,E2 -17784.618} C_VEL
LIN {X 0,Y 311.51,Z 580.777,A -85,B 0,C 180,E1 -17785.665,E2 -17785.665} C_VEL
LIN {X 0,Y 306.815,Z 595.112,A -85,B 0,C 180,E1 -17787.042,E2 -17787.042} C_VEL
LIN {X 0,Y 301.953,Z 608.293,A -85,B 0,C 180,E1 -17788.615,E2 -17788.615} C_VEL
LIN {X 0,Y 296.682,Z 621.332,A -85,B 0,C 180,E1 -17790.558,E2 -17790.558} C_VEL
LIN {X 0,Y 292.302,Z 631.477,A -85,B 0,C 180,E1 -17792.43,E2 -17792.43} C_VEL
LIN {X 0,Y 287.907,Z 641.067,A -85,B 0,C 180,E1 -17794.582,E2 -17794.582} C_VEL
LIN {X 0,Y 283.62,Z 649.918,A -85,B 0,C 180,E1 -17797.028,E2 -17797.028} C_VEL
LIN {X 0,Y 279.894,Z 656.917,A -85,B 0,C 180,E1 -17799.419,E2 -17799.419} C_VEL
LIN {X 0,Y 276.507,Z 663.262,A -85,B 0,C 180,E1 -17802.242,E2 -17802.242} C_VEL
LIN {X 0,Y 273.724,Z 668.09,A -85,B 0,C 180,E1 -17805.123,E2 -17805.123} C_VEL
LIN {X 0,Y 271.755,Z 671.463,A -85,B 0,C 180,E1 -17808.06,E2 -17808.06} C_VEL
LIN {X 0,Y 270.113,Z 673.502,A -85,B 0,C 180,E1 -17811.019,E2 -17811.019} C_VEL
LIN {X 0,Y 269.12,Z 674.171,A -85,B 0,C 180,E1 -17814.004,E2 -17814.004} C_VEL
LIN {X 0,Y 268.605,Z 673.464,A -85,B 0,C 180,E1 -17817.001,E2 -17817.001} C_VEL
LIN {X 0,Y 268.328,Z 671.362,A -85,B 0,C 180,E1 -17820,E2 -17820} C_VEL
LIN {X 0,Y 268.381,Z 667.795,A -85,B 0,C 180,E1 -17823.002,E2 -17823.002} C_VEL
LIN {X 0,Y 268.541,Z 662.663,A -85,B 0,C 180,E1 -17826.009,E2 -17826.009} C_VEL
LIN {X 0,Y 268.839,Z 657.622,A -85,B 0,C 180,E1 -17828.267,E2 -17828.267} C_VEL
LIN {X 0,Y 269.442,Z 650.397,A -85,B 0,C 180,E1 -17830.901,E2 -17830.901} C_VEL
LIN {X 0,Y 270.332,Z 641.469,A -85,B 0,C 180,E1 -17833.532,E2 -17833.532} C_VEL
LIN {X 0,Y 271.424,Z 632.158,A -85,B 0,C 180,E1 -17835.776,E2 -17835.776} C_VEL
LIN {X 0,Y 272.519,Z 622.198,A -85,B 0,C 180,E1 -17837.792,E2 -17837.792} C_VEL
LIN {X 0,Y 273.962,Z 609.815,A -85,B 0,C 180,E1 -17839.871,E2 -17839.871} C_VEL
LIN {X 0,Y 275.538,Z 596.501,A -85,B 0,C 180,E1 -17841.706,E2 -17841.706} C_VEL
LIN {X 0,Y 276.967,Z 583.56,A -85,B 0,C 180,E1 -17843.161,E2 -17843.161} C_VEL
LIN {X 0,Y 278.199,Z 570.591,A -85,B 0,C 180,E1 -17844.342,E2 -17844.342} C_VEL
LIN {X 0,Y 279.499,Z 554.761,A -85,B 0,C 180,E1 -17845.457,E2 -17845.457} C_VEL
LIN {X 0,Y 280.647,Z 538.124,A -85,B 0,C 180,E1 -17846.291,E2 -17846.291} C_VEL
LIN {X 0,Y 286.11,Z 441.725,A -85,B 0,C 180,E1 -17850.004,E2 -17850.004} C_VEL
LIN {X 0,Y 282.29,Z 414.582,A -85,B 0,C 180,E1 -17851.433,E2 -17851.433} C_VEL
LIN {X 0,Y 276.618,Z 398.438,A -85,B 0,C 180,E1 -17852.61,E2 -17852.61} C_VEL
LIN {X 0,Y 274.079,Z 387.272,A -85,B 0,C 180,E1 -17855.772,E2 -17855.772} C_VEL
LIN {X 0,Y 271.017,Z 374.69,A -85,B 0,C 180,E1 -17859.663,E2 -17859.663} C_VEL
LIN {X 0,Y 271.171,Z 374.703,A -85,B 0,C 180,E1 -17859.985,E2 -17859.985} C_VEL
LIN {X 0,Y 271.727,Z 375.332,A -85,B 0,C 180,E1 -17860.286,E2 -17860.286} C_VEL
LIN {X 0,Y 275.663,Z 385.068,A -85,B 0,C 180,E1 -17863.501,E2 -17863.501} C_VEL
LIN {X 0,Y 278.781,Z 393.214,A -85,B 0,C 180,E1 -17865.929,E2 -17865.929} C_VEL
LIN {X 0,Y 279.788,Z 395.933,A -85,B 0,C 180,E1 -17866.654,E2 -17866.654} C_VEL
LIN {X 0,Y 288.946,Z 412.154,A -85,B 0,C 180,E1 -17868.874,E2 -17868.874} C_VEL
LIN {X 0,Y 296.531,Z 427.598,A -85,B 0,C 180,E1 -17870.612,E2 -17870.612} C_VEL
LIN {X 0,Y 300.81,Z 437.867,A -85,B 0,C 180,E1 -17871.583,E2 -17871.583} C_VEL
LIN {X 0,Y 302.627,Z 450.337,A -85,B 0,C 180,E1 -17872.222,E2 -17872.222} C_VEL
LIN {X 0,Y 298.311,Z 552.241,A -85,B 0,C 180,E1 -17874.591,E2 -17874.591} C_VEL
LIN {X 0,Y 297.321,Z 569.7,A -85,B 0,C 180,E1 -17875.077,E2 -17875.077} C_VEL
LIN {X 0,Y 295.717,Z 584.982,A -85,B 0,C 180,E1 -17875.739,E2 -17875.739} C_VEL
LIN {X 0,Y 293.78,Z 599.209,A -85,B 0,C 180,E1 -17876.618,E2 -17876.618} C_VEL
LIN {X 0,Y 291.414,Z 613.336,A -85,B 0,C 180,E1 -17877.77,E2 -17877.77} C_VEL
LIN {X 0,Y 288.572,Z 627.437,A -85,B 0,C 180,E1 -17879.24,E2 -17879.24} C_VEL
LIN {X 0,Y 285.596,Z 640.337,A -85,B 0,C 180,E1 -17880.921,E2 -17880.921} C_VEL
LIN {X 0,Y 282.815,Z 651.177,A -85,B 0,C 180,E1 -17882.63,E2 -17882.63} C_VEL
LIN {X 0,Y 279.836,Z 662.138,A -85,B 0,C 180,E1 -17884.726,E2 -17884.726} C_VEL
LIN {X 0,Y 277.381,Z 671.367,A -85,B 0,C 180,E1 -17886.876,E2 -17886.876} C_VEL
LIN {X 0,Y 274.709,Z 680.439,A -85,B 0,C 180,E1 -17889.404,E2 -17889.404} C_VEL
LIN {X 0,Y 272.264,Z 689.051,A -85,B 0,C 180,E1 -17892.375,E2 -17892.375} C_VEL
LIN {X 0,Y 270.742,Z 694.999,A -85,B 0,C 180,E1 -17894.954,E2 -17894.954} C_VEL
LIN {X 0,Y 269.394,Z 700.526,A -85,B 0,C 180,E1 -17897.953,E2 -17897.953} C_VEL
LIN {X 0,Y 268.642,Z 704.709,A -85,B 0,C 180,E1 -17900.969,E2 -17900.969} C_VEL
LIN {X 0,Y 268.217,Z 707.647,A -85,B 0,C 180,E1 -17903.984,E2 -17903.984} C_VEL
LIN {X 0,Y 268.101,Z 709.407,A -85,B 0,C 180,E1 -17906.995,E2 -17906.995} C_VEL
LIN {X 0,Y 268.128,Z 710.016,A -85,B 0,C 180,E1 -17910,E2 -17910} C_VEL
LIN {X 0,Y 268.102,Z 709.442,A -85,B 0,C 180,E1 -17913.005,E2 -17913.005} C_VEL
LIN {X 0,Y 268.221,Z 707.729,A -85,B 0,C 180,E1 -17916.016,E2 -17916.016} C_VEL
LIN {X 0,Y 268.641,Z 704.845,A -85,B 0,C 180,E1 -17919.031,E2 -17919.031} C_VEL
LIN {X 0,Y 269.367,Z 700.721,A -85,B 0,C 180,E1 -17922.048,E2 -17922.048} C_VEL
LIN {X 0,Y 270.703,Z 695.246,A -85,B 0,C 180,E1 -17925.047,E2 -17925.047} C_VEL
LIN {X 0,Y 272.508,Z 688.274,A -85,B 0,C 180,E1 -17928.028,E2 -17928.028} C_VEL
LIN {X 0,Y 274.615,Z 680.81,A -85,B 0,C 180,E1 -17930.603,E2 -17930.603} C_VEL
LIN {X 0,Y 277.296,Z 671.817,A -85,B 0,C 180,E1 -17933.131,E2 -17933.131} C_VEL
LIN {X 0,Y 280.207,Z 660.943,A -85,B 0,C 180,E1 -17935.636,E2 -17935.636} C_VEL
LIN {X 0,Y 283.256,Z 649.773,A -85,B 0,C 180,E1 -17937.724,E2 -17937.724} C_VEL
LIN {X 0,Y 286.335,Z 637.504,A -85,B 0,C 180,E1 -17939.601,E2 -17939.601} C_VEL
LIN {X 0,Y 289.399,Z 623.95,A -85,B 0,C 180,E1 -17941.271,E2 -17941.271} C_VEL
LIN {X 0,Y 292.083,Z 609.884,A -85,B 0,C 180,E1 -17942.656,E2 -17942.656} C_VEL
LIN {X 0,Y 294.27,Z 595.987,A -85,B 0,C 180,E1 -17943.73,E2 -17943.73} C_VEL
LIN {X 0,Y 296.202,Z 581.478,A -85,B 0,C 180,E1 -17944.557,E2 -17944.557} C_VEL
LIN {X 0,Y 297.599,Z 566.813,A -85,B 0,C 180,E1 -17945.144,E2 -17945.144} C_VEL
LIN {X 0,Y 299.375,Z 529.114,A -85,B 0,C 180,E1 -17946.059,E2 -17946.059} C_VEL
LIN {X 0,Y 301.281,Z 483.273,A -85,B 0,C 180,E1 -17947.129,E2 -17947.129} C_VEL
LIN {X 0,Y 300.99,Z 477.474,A -85,B 0,C 180,E1 -17947.341,E2 -17947.341} C_VEL
LIN {X 0,Y 297.212,Z 458.88,A -85,B 0,C 180,E1 -17948.456,E2 -17948.456} C_VEL
LIN {X 0,Y 297.028,Z 453.08,A -85,B 0,C 180,E1 -17948.66,E2 -17948.66} C_VEL
LIN {X 0,Y 296.966,Z 449.915,A -85,B 0,C 180,E1 -17948.766,E2 -17948.766} C_VEL
LIN {X 0,Y 295.225,Z 439.626,A -85,B 0,C 180,E1 -17949.352,E2 -17949.352} C_VEL
LIN {X 0,Y 289.171,Z 426.066,A -85,B 0,C 180,E1 -17950.772,E2 -17950.772} C_VEL
LIN {X 0,Y 282.45,Z 412.831,A -85,B 0,C 180,E1 -17952.396,E2 -17952.396} C_VEL
LIN {X 0,Y 273.849,Z 397.908,A -85,B 0,C 180,E1 -17954.588,E2 -17954.588} C_VEL
LIN {X 0,Y 272.348,Z 395.211,A -85,B 0,C 180,E1 -17955.055,E2 -17955.055} C_VEL
LIN {X 0,Y 268.248,Z 384.676,A -85,B 0,C 180,E1 -17958.382,E2 -17958.382} C_VEL
LIN {X 0,Y 264.674,Z 376.03,A -85,B 0,C 180,E1 -17961.415,E2 -17961.415} C_VEL
LIN {X 0,Y 263.243,Z 372.884,A -85,B 0,C 180,E1 -17962.642,E2 -17962.642} C_VEL
LIN {X 0,Y 263.164,Z 372.336,A -85,B 0,C 180,E1 -17963.087,E2 -17963.087} C_VEL
LIN {X 0,Y 263.151,Z 372.326,A -85,B 0,C 180,E1 -17965.885,E2 -17965.885} C_VEL
LIN {X 0,Y 263.126,Z 372.322,A -85,B 0,C 180,E1 -17969.503,E2 -17969.503} C_VEL
LIN {X 0,Y 263.141,Z 372.312,A -85,B 0,C 180,E1 -17972.997,E2 -17972.997} C_VEL
LIN {X 0,Y 263.144,Z 372.319,A -85,B 0,C 180,E1 -17976.383,E2 -17976.383} C_VEL
LIN {X 0,Y 263.243,Z 372.313,A -85,B 0,C 180,E1 -17979.692,E2 -17979.692} C_VEL
LIN {X 0,Y 263.324,Z 372.292,A -85,B 0,C 180,E1 -17984.52,E2 -17984.52} C_VEL
LIN {X 0,Y 263.35,Z 372.278,A -85,B 0,C 180,E1 -17989.233,E2 -17989.233} C_VEL
LIN {X 0,Y 263.545,Z 372.282,A -85,B 0,C 180,E1 -17992.337,E2 -17992.337} C_VEL
LIN {X 0,Y 263.748,Z 372.257,A -85,B 0,C 180,E1 -17998.473,E2 -17998.473} C_VEL
LIN {X 0,Y 263.749,Z 372.226,A -85,B 0,C 180,E1 -18001.527,E2 -18001.527} C_VEL
LIN {X 0,Y 263.529,Z 372.252,A -85,B 0,C 180,E1 -18007.663,E2 -18007.663} C_VEL
LIN {X 0,Y 263.35,Z 372.304,A -85,B 0,C 180,E1 -18010.766,E2 -18010.766} C_VEL
LIN {X 0,Y 263.315,Z 372.294,A -85,B 0,C 180,E1 -18015.48,E2 -18015.48} C_VEL
LIN {X 0,Y 263.252,Z 372.295,A -85,B 0,C 180,E1 -18020.307,E2 -18020.307} C_VEL
LIN {X 0,Y 263.209,Z 372.302,A -85,B 0,C 180,E1 -18025.291,E2 -18025.291} C_VEL
LIN {X 0,Y 263.166,Z 372.316,A -85,B 0,C 180,E1 -18028.731,E2 -18028.731} C_VEL
LIN {X 0,Y 263.133,Z 372.336,A -85,B 0,C 180,E1 -18032.288,E2 -18032.288} C_VEL
LIN {X 0,Y 263.181,Z 372.325,A -85,B 0,C 180,E1 -18036.763,E2 -18036.763} C_VEL
LIN {X 0,Y 263.151,Z 372.503,A -85,B 0,C 180,E1 -18039.989,E2 -18039.989} C_VEL
LIN {X 0,Y 263.314,Z 373.281,A -85,B 0,C 180,E1 -18040.334,E2 -18040.334} C_VEL
LIN {X 0,Y 264.769,Z 376.01,A -85,B 0,C 180,E1 -18041.155,E2 -18041.155} C_VEL
LIN {X 0,Y 265.446,Z 376.816,A -85,B 0,C 180,E1 -18041.445,E2 -18041.445} C_VEL
LIN {X 0,Y 274.093,Z 392.612,A -85,B 0,C 180,E1 -18045.586,E2 -18045.586} C_VEL
LIN {X 0,Y 278.69,Z 400.038,A -85,B 0,C 180,E1 -18046.77,E2 -18046.77} C_VEL
LIN {X 0,Y 287.312,Z 418.615,A -85,B 0,C 180,E1 -18048.979,E2 -18048.979} C_VEL
LIN {X 0,Y 295.516,Z 438.017,A -85,B 0,C 180,E1 -18050.953,E2 -18050.953} C_VEL
LIN {X 0,Y 296.624,Z 447.773,A -85,B 0,C 180,E1 -18051.424,E2 -18051.424} C_VEL
LIN {X 0,Y 291.397,Z 564.795,A -85,B 0,C 180,E1 -18054.206,E2 -18054.206} C_VEL
LIN {X 0,Y 289.981,Z 580.169,A -85,B 0,C 180,E1 -18054.805,E2 -18054.805} C_VEL
LIN {X 0,Y 288.247,Z 593.706,A -85,B 0,C 180,E1 -18055.573,E2 -18055.573} C_VEL
LIN {X 0,Y 286.148,Z 606.547,A -85,B 0,C 180,E1 -18056.523,E2 -18056.523} C_VEL
LIN {X 0,Y 283.654,Z 620.059,A -85,B 0,C 180,E1 -18057.812,E2 -18057.812} C_VEL
LIN {X 0,Y 280.733,Z 632.956,A -85,B 0,C 180,E1 -18059.331,E2 -18059.331} C_VEL
LIN {X 0,Y 277.773,Z 644.844,A -85,B 0,C 180,E1 -18061.061,E2 -18061.061} C_VEL
LIN {X 0,Y 274.747,Z 655.833,A -85,B 0,C 180,E1 -18062.997,E2 -18062.997} C_VEL
LIN {X 0,Y 271.85,Z 666.403,A -85,B 0,C 180,E1 -18065.282,E2 -18065.282} C_VEL
LIN {X 0,Y 268.966,Z 675.808,A -85,B 0,C 180,E1 -18067.736,E2 -18067.736} C_VEL
LIN {X 0,Y 266.57,Z 683.984,A -85,B 0,C 180,E1 -18070.358,E2 -18070.358} C_VEL
LIN {X 0,Y 264.595,Z 690.744,A -85,B 0,C 180,E1 -18073.012,E2 -18073.012} C_VEL
LIN {X 0,Y 263.028,Z 697.004,A -85,B 0,C 180,E1 -18076.086,E2 -18076.086} C_VEL
LIN {X 0,Y 261.929,Z 701.831,A -85,B 0,C 180,E1 -18079.175,E2 -18079.175} C_VEL
LIN {X 0,Y 261.306,Z 705.359,A -85,B 0,C 180,E1 -18082.272,E2 -18082.272} C_VEL
LIN {X 0,Y 261.045,Z 707.68,A -85,B 0,C 180,E1 -18085.368,E2 -18085.368} C_VEL
LIN {X 0,Y 261.044,Z 708.845,A -85,B 0,C 180,E1 -18088.457,E2 -18088.457} C_VEL
LIN {X 0,Y 261.045,Z 708.842,A -85,B 0,C 180,E1 -18091.543,E2 -18091.543} C_VEL
LIN {X 0,Y 261.048,Z 707.454,A -85,B 0,C 180,E1 -18095.048,E2 -18095.048} C_VEL
LIN {X 0,Y 261.307,Z 705.336,A -85,B 0,C 180,E1 -18097.729,E2 -18097.729} C_VEL
LIN {X 0,Y 261.93,Z 701.789,A -85,B 0,C 180,E1 -18100.826,E2 -18100.826} C_VEL
LIN {X 0,Y 263.035,Z 696.945,A -85,B 0,C 180,E1 -18103.914,E2 -18103.914} C_VEL
LIN {X 0,Y 264.659,Z 690.495,A -85,B 0,C 180,E1 -18107.065,E2 -18107.065} C_VEL
LIN {X 0,Y 266.887,Z 682.795,A -85,B 0,C 180,E1 -18110.019,E2 -18110.019} C_VEL
LIN {X 0,Y 268.335,Z 678.998,A -85,B 0,C 180,E1 -18111.511,E2 -18111.511} C_VEL
LIN {X 0,Y 271.969,Z 671.516,A -85,B 0,C 180,E1 -18114.423,E2 -18114.423} C_VEL
LIN {X 0,Y 276.361,Z 662.489,A -85,B 0,C 180,E1 -18117.242,E2 -18117.242} C_VEL
LIN {X 0,Y 280.926,Z 653.115,A -85,B 0,C 180,E1 -18119.61,E2 -18119.61} C_VEL
LIN {X 0,Y 286.06,Z 642.171,A -85,B 0,C 180,E1 -18121.885,E2 -18121.885} C_VEL
LIN {X 0,Y 291.902,Z 629.292,A -85,B 0,C 180,E1 -18124.041,E2 -18124.041} C_VEL
LIN {X 0,Y 297.37,Z 616.311,A -85,B 0,C 180,E1 -18125.799,E2 -18125.799} C_VEL
LIN {X 0,Y 302.855,Z 602.191,A -85,B 0,C 180,E1 -18127.319,E2 -18127.319} C_VEL
LIN {X 0,Y 307.683,Z 588.502,A -85,B 0,C 180,E1 -18128.494,E2 -18128.494} C_VEL
LIN {X 0,Y 313.167,Z 570.735,A -85,B 0,C 180,E1 -18129.657,E2 -18129.657} C_VEL
LIN {X 0,Y 317.478,Z 553.858,A -85,B 0,C 180,E1 -18130.458,E2 -18130.458} C_VEL
LIN {X 0,Y 333.044,Z 481.883,A -85,B 0,C 180,E1 -18133.316,E2 -18133.316} C_VEL
LIN {X 0,Y 334.767,Z 474.371,A -85,B 0,C 180,E1 -18133.624,E2 -18133.624} C_VEL
LIN {X 0,Y 334.434,Z 473.107,A -85,B 0,C 180,E1 -18134.584,E2 -18134.584} C_VEL
LIN {X 0,Y 334.03,Z 472.718,A -85,B 0,C 180,E1 -18136.027,E2 -18136.027} C_VEL
LIN {X 0,Y 334.211,Z 473.261,A -85,B 0,C 180,E1 -18138.08,E2 -18138.08} C_VEL
LIN {X 0,Y 334.443,Z 475.194,A -85,B 0,C 180,E1 -18139.259,E2 -18139.259} C_VEL
LIN {X 0,Y 316.43,Z 554.378,A -85,B 0,C 180,E1 -18142.655,E2 -18142.655} C_VEL
LIN {X 0,Y 312.742,Z 567.952,A -85,B 0,C 180,E1 -18143.451,E2 -18143.451} C_VEL
LIN {X 0,Y 308.464,Z 581.572,A -85,B 0,C 180,E1 -18144.48,E2 -18144.48} C_VEL
LIN {X 0,Y 303.001,Z 596.915,A -85,B 0,C 180,E1 -18145.974,E2 -18145.974} C_VEL
LIN {X 0,Y 297.404,Z 610.75,A -85,B 0,C 180,E1 -18147.68,E2 -18147.68} C_VEL
LIN {X 0,Y 291.877,Z 623.339,A -85,B 0,C 180,E1 -18149.626,E2 -18149.626} C_VEL
LIN {X 0,Y 287.232,Z 633.16,A -85,B 0,C 180,E1 -18151.502,E2 -18151.502} C_VEL
LIN {X 0,Y 282.378,Z 642.837,A -85,B 0,C 180,E1 -18153.767,E2 -18153.767} C_VEL
LIN {X 0,Y 277.977,Z 651.037,A -85,B 0,C 180,E1 -18156.139,E2 -18156.139} C_VEL
LIN {X 0,Y 273.473,Z 658.715,A -85,B 0,C 180,E1 -18158.913,E2 -18158.913} C_VEL
LIN {X 0,Y 269.9,Z 664.721,A -85,B 0,C 180,E1 -18161.792,E2 -18161.792} C_VEL
LIN {X 0,Y 266.973,Z 669.255,A -85,B 0,C 180,E1 -18164.737,E2 -18164.737} C_VEL
LIN {X 0,Y 264.866,Z 672.368,A -85,B 0,C 180,E1 -18167.745,E2 -18167.745} C_VEL
LIN {X 0,Y 263.149,Z 674.165,A -85,B 0,C 180,E1 -18170.779,E2 -18170.779} C_VEL
LIN {X 0,Y 262.075,Z 674.609,A -85,B 0,C 180,E1 -18173.842,E2 -18173.842} C_VEL
LIN {X 0,Y 261.536,Z 673.687,A -85,B 0,C 180,E1 -18176.919,E2 -18176.919} C_VEL
LIN {X 0,Y 261.249,Z 671.381,A -85,B 0,C 180,E1 -18180,E2 -18180} C_VEL
LIN {X 0,Y 261.292,Z 667.605,A -85,B 0,C 180,E1 -18183.084,E2 -18183.084} C_VEL
LIN {X 0,Y 261.442,Z 662.674,A -85,B 0,C 180,E1 -18185.942,E2 -18185.942} C_VEL
LIN {X 0,Y 261.858,Z 656.021,A -85,B 0,C 180,E1 -18188.878,E2 -18188.878} C_VEL
LIN {X 0,Y 262.528,Z 648.303,A -85,B 0,C 180,E1 -18191.583,E2 -18191.583} C_VEL
LIN {X 0,Y 263.548,Z 638.789,A -85,B 0,C 180,E1 -18194.281,E2 -18194.281} C_VEL
LIN {X 0,Y 264.63,Z 628.902,A -85,B 0,C 180,E1 -18196.589,E2 -18196.589} C_VEL
LIN {X 0,Y 266.125,Z 617.021,A -85,B 0,C 180,E1 -18198.875,E2 -18198.875} C_VEL
LIN {X 0,Y 267.649,Z 603.742,A -85,B 0,C 180,E1 -18200.963,E2 -18200.963} C_VEL
LIN {X 0,Y 269.293,Z 590.643,A -85,B 0,C 180,E1 -18202.64,E2 -18202.64} C_VEL
LIN {X 0,Y 270.826,Z 576.318,A -85,B 0,C 180,E1 -18204.124,E2 -18204.124} C_VEL
LIN {X 0,Y 272.028,Z 562.19,A -85,B 0,C 180,E1 -18205.278,E2 -18205.278} C_VEL
LIN {X 0,Y 273.269,Z 545.688,A -85,B 0,C 180,E1 -18206.285,E2 -18206.285} C_VEL
LIN {X 0,Y 276.043,Z 497.861,A -85,B 0,C 180,E1 -18208.255,E2 -18208.255} C_VEL
LIN {X 0,Y 279.282,Z 441.955,A -85,B 0,C 180,E1 -18210.472,E2 -18210.472} C_VEL
LIN {X 0,Y 275.714,Z 416.464,A -85,B 0,C 180,E1 -18211.859,E2 -18211.859} C_VEL
LIN {X 0,Y 269.323,Z 398.284,A -85,B 0,C 180,E1 -18213.23,E2 -18213.23} C_VEL
LIN {X 0,Y 266.753,Z 387.066,A -85,B 0,C 180,E1 -18216.529,E2 -18216.529} C_VEL
LIN {X 0,Y 264.754,Z 378.87,A -85,B 0,C 180,E1 -18219.135,E2 -18219.135} C_VEL
LIN {X 0,Y 265.018,Z 378.887,A -85,B 0,C 180,E1 -18219.528,E2 -18219.528} C_VEL
LIN {X 0,Y 266.099,Z 379.665,A -85,B 0,C 180,E1 -18220.01,E2 -18220.01} C_VEL
LIN {X 0,Y 270.07,Z 389.22,A -85,B 0,C 180,E1 -18223.227,E2 -18223.227} C_VEL
LIN {X 0,Y 272.454,Z 395.417,A -85,B 0,C 180,E1 -18225.138,E2 -18225.138} C_VEL
LIN {X 0,Y 280.926,Z 410.072,A -85,B 0,C 180,E1 -18227.364,E2 -18227.364} C_VEL
LIN {X 0,Y 288.153,Z 424.001,A -85,B 0,C 180,E1 -18229.12,E2 -18229.12} C_VEL
LIN {X 0,Y 295.037,Z 439.381,A -85,B 0,C 180,E1 -18230.739,E2 -18230.739} C_VEL
LIN {X 0,Y 295.747,Z 442.279,A -85,B 0,C 180,E1 -18230.94,E2 -18230.94} C_VEL
LIN {X 0,Y 297.005,Z 451.057,A -85,B 0,C 180,E1 -18231.402,E2 -18231.402} C_VEL
LIN {X 0,Y 292.441,Z 553.923,A -85,B 0,C 180,E1 -18233.822,E2 -18233.822} C_VEL
LIN {X 0,Y 291.424,Z 570.705,A -85,B 0,C 180,E1 -18234.316,E2 -18234.316} C_VEL
LIN {X 0,Y 289.795,Z 585.669,A -85,B 0,C 180,E1 -18234.991,E2 -18234.991} C_VEL
LIN {X 0,Y 287.712,Z 600.183,A -85,B 0,C 180,E1 -18235.915,E2 -18235.915} C_VEL
LIN {X 0,Y 285.115,Z 614.879,A -85,B 0,C 180,E1 -18237.16,E2 -18237.16} C_VEL
LIN {X 0,Y 282.151,Z 628.809,A -85,B 0,C 180,E1 -18238.67,E2 -18238.67} C_VEL
LIN {X 0,Y 279.09,Z 641.469,A -85,B 0,C 180,E1 -18240.383,E2 -18240.383} C_VEL
LIN {X 0,Y 275.954,Z 653.081,A -85,B 0,C 180,E1 -18242.303,E2 -18242.303} C_VEL
LIN {X 0,Y 272.897,Z 663.912,A -85,B 0,C 180,E1 -18244.492,E2 -18244.492} C_VEL
LIN {X 0,Y 270.373,Z 672.756,A -85,B 0,C 180,E1 -18246.646,E2 -18246.646} C_VEL
LIN {X 0,Y 267.665,Z 681.607,A -85,B 0,C 180,E1 -18249.239,E2 -18249.239} C_VEL
LIN {X 0,Y 265.195,Z 689.884,A -85,B 0,C 180,E1 -18252.257,E2 -18252.257} C_VEL
LIN {X 0,Y 263.472,Z 696.516,A -85,B 0,C 180,E1 -18255.32,E2 -18255.32} C_VEL
LIN {X 0,Y 262.161,Z 701.708,A -85,B 0,C 180,E1 -18258.401,E2 -18258.401} C_VEL
LIN {X 0,Y 261.583,Z 704.695,A -85,B 0,C 180,E1 -18260.723,E2 -18260.723} C_VEL
LIN {X 0,Y 261.144,Z 707.634,A -85,B 0,C 180,E1 -18263.82,E2 -18263.82} C_VEL
LIN {X 0,Y 260.999,Z 709.394,A -85,B 0,C 180,E1 -18266.913,E2 -18266.913} C_VEL
LIN {X 0,Y 261.035,Z 710.003,A -85,B 0,C 180,E1 -18270,E2 -18270} C_VEL
LIN {X 0,Y 261.001,Z 709.428,A -85,B 0,C 180,E1 -18273.087,E2 -18273.087} C_VEL
LIN {X 0,Y 261.146,Z 707.715,A -85,B 0,C 180,E1 -18276.18,E2 -18276.18} C_VEL
LIN {X 0,Y 261.58,Z 704.83,A -85,B 0,C 180,E1 -18279.277,E2 -18279.277} C_VEL
LIN {X 0,Y 262.378,Z 700.705,A -85,B 0,C 180,E1 -18282.373,E2 -18282.373} C_VEL
LIN {X 0,Y 263.787,Z 695.23,A -85,B 0,C 180,E1 -18285.452,E2 -18285.452} C_VEL
LIN {X 0,Y 265.696,Z 688.256,A -85,B 0,C 180,E1 -18288.506,E2 -18288.506} C_VEL
LIN {X 0,Y 267.935,Z 680.791,A -85,B 0,C 180,E1 -18291.141,E2 -18291.141} C_VEL
LIN {X 0,Y 270.738,Z 671.797,A -85,B 0,C 180,E1 -18293.726,E2 -18293.726} C_VEL
LIN {X 0,Y 273.3,Z 662.606,A -85,B 0,C 180,E1 -18295.923,E2 -18295.923} C_VEL
LIN {X 0,Y 276.399,Z 651.742,A -85,B 0,C 180,E1 -18298.06,E2 -18298.06} C_VEL
LIN {X 0,Y 279.547,Z 639.866,A -85,B 0,C 180,E1 -18299.978,E2 -18299.978} C_VEL
LIN {X 0,Y 282.716,Z 626.855,A -85,B 0,C 180,E1 -18301.678,E2 -18301.678} C_VEL
LIN {X 0,Y 285.576,Z 612.868,A -85,B 0,C 180,E1 -18303.15,E2 -18303.15} C_VEL
LIN {X 0,Y 288.05,Z 598.303,A -85,B 0,C 180,E1 -18304.348,E2 -18304.348} C_VEL
LIN {X 0,Y 290.188,Z 583.048,A -85,B 0,C 180,E1 -18305.272,E2 -18305.272} C_VEL
LIN {X 0,Y 291.743,Z 567.916,A -85,B 0,C 180,E1 -18305.904,E2 -18305.904} C_VEL
LIN {X 0,Y 292.861,Z 545.675,A -85,B 0,C 180,E1 -18306.491,E2 -18306.491} C_VEL
LIN {X 0,Y 296.307,Z 468.176,A -85,B 0,C 180,E1 -18308.312,E2 -18308.312} C_VEL
LIN {X 0,Y 297.028,Z 453.08,A -85,B 0,C 180,E1 -18308.66,E2 -18308.66} C_VEL
LIN {X 0,Y 296.749,Z 449.338,A -85,B 0,C 180,E1 -18308.817,E2 -18308.817} C_VEL
LIN {X 0,Y 295.299,Z 445.077,A -85,B 0,C 180,E1 -18309.173,E2 -18309.173} C_VEL
LIN {X 0,Y 292.094,Z 439.949,A -85,B 0,C 180,E1 -18309.845,E2 -18309.845} C_VEL
LIN {X 0,Y 285.469,Z 431.577,A -85,B 0,C 180,E1 -18311.231,E2 -18311.231} C_VEL
LIN {X 0,Y 283.635,Z 428.413,A -85,B 0,C 180,E1 -18311.66,E2 -18311.66} C_VEL
LIN {X 0,Y 276.388,Z 414.262,A -85,B 0,C 180,E1 -18313.498,E2 -18313.498} C_VEL
LIN {X 0,Y 269.561,Z 402.424,A -85,B 0,C 180,E1 -18315.32,E2 -18315.32} C_VEL
LIN {X 0,Y 265.218,Z 395.312,A -85,B 0,C 180,E1 -18316.582,E2 -18316.582} C_VEL
LIN {X 0,Y 261.363,Z 385.654,A -85,B 0,C 180,E1 -18319.808,E2 -18319.808} C_VEL
LIN {X 0,Y 257.644,Z 376.77,A -85,B 0,C 180,E1 -18323.122,E2 -18323.122} C_VEL
LIN {X 0,Y 256.138,Z 373.507,A -85,B 0,C 180,E1 -18324.515,E2 -18324.515} C_VEL
LIN {X 0,Y 256.104,Z 373.198,A -85,B 0,C 180,E1 -18325.412,E2 -18325.412} C_VEL
LIN {X 0,Y 256.083,Z 373.194,A -85,B 0,C 180,E1 -18328.571,E2 -18328.571} C_VEL
LIN {X 0,Y 256.093,Z 373.192,A -85,B 0,C 180,E1 -18332.19,E2 -18332.19} C_VEL
LIN {X 0,Y 256.133,Z 373.203,A -85,B 0,C 180,E1 -18335.695,E2 -18335.695} C_VEL
LIN {X 0,Y 256.146,Z 373.187,A -85,B 0,C 180,E1 -18339.103,E2 -18339.103} C_VEL
LIN {X 0,Y 256.229,Z 373.168,A -85,B 0,C 180,E1 -18343.739,E2 -18343.739} C_VEL
LIN {X 0,Y 256.26,Z 373.175,A -85,B 0,C 180,E1 -18347.326,E2 -18347.326} C_VEL
LIN {X 0,Y 256.435,Z 373.15,A -85,B 0,C 180,E1 -18350.622,E2 -18350.622} C_VEL
LIN {X 0,Y 256.473,Z 373.143,A -85,B 0,C 180,E1 -18353.707,E2 -18353.707} C_VEL
LIN {X 0,Y 256.71,Z 373.134,A -85,B 0,C 180,E1 -18358.431,E2 -18358.431} C_VEL
LIN {X 0,Y 256.712,Z 373.102,A -85,B 0,C 180,E1 -18361.569,E2 -18361.569} C_VEL
LIN {X 0,Y 256.461,Z 373.143,A -85,B 0,C 180,E1 -18366.293,E2 -18366.293} C_VEL
LIN {X 0,Y 256.427,Z 373.15,A -85,B 0,C 180,E1 -18369.465,E2 -18369.465} C_VEL
LIN {X 0,Y 256.235,Z 373.163,A -85,B 0,C 180,E1 -18374.291,E2 -18374.291} C_VEL
LIN {X 0,Y 256.18,Z 373.193,A -85,B 0,C 180,E1 -18377.564,E2 -18377.564} C_VEL
LIN {X 0,Y 256.153,Z 373.187,A -85,B 0,C 180,E1 -18381.117,E2 -18381.117} C_VEL
LIN {X 0,Y 256.189,Z 373.175,A -85,B 0,C 180,E1 -18385.138,E2 -18385.138} C_VEL
LIN {X 0,Y 256.104,Z 373.189,A -85,B 0,C 180,E1 -18389.601,E2 -18389.601} C_VEL
LIN {X 0,Y 256.067,Z 373.202,A -85,B 0,C 180,E1 -18393.293,E2 -18393.293} C_VEL
LIN {X 0,Y 256.128,Z 373.209,A -85,B 0,C 180,E1 -18397.879,E2 -18397.879} C_VEL
LIN {X 0,Y 256.194,Z 373.762,A -85,B 0,C 180,E1 -18398.365,E2 -18398.365} C_VEL
LIN {X 0,Y 257.682,Z 376.843,A -85,B 0,C 180,E1 -18399.365,E2 -18399.365} C_VEL
LIN {X 0,Y 260.909,Z 382.016,A -85,B 0,C 180,E1 -18401.043,E2 -18401.043} C_VEL
LIN {X 0,Y 266.476,Z 392.513,A -85,B 0,C 180,E1 -18403.944,E2 -18403.944} C_VEL
LIN {X 0,Y 273.12,Z 402.273,A -85,B 0,C 180,E1 -18405.735,E2 -18405.735} C_VEL
LIN {X 0,Y 277.369,Z 410.923,A -85,B 0,C 180,E1 -18406.891,E2 -18406.891} C_VEL
LIN {X 0,Y 284.889,Z 427.923,A -85,B 0,C 180,E1 -18408.857,E2 -18408.857} C_VEL
LIN {X 0,Y 290.189,Z 440.738,A -85,B 0,C 180,E1 -18410.176,E2 -18410.176} C_VEL
LIN {X 0,Y 291.097,Z 448.485,A -85,B 0,C 180,E1 -18410.569,E2 -18410.569} C_VEL
LIN {X 0,Y 285.67,Z 564.912,A -85,B 0,C 180,E1 -18413.374,E2 -18413.374} C_VEL
LIN {X 0,Y 284.23,Z 580.242,A -85,B 0,C 180,E1 -18413.983,E2 -18413.983} C_VEL
LIN {X 0,Y 282.411,Z 593.76,A -85,B 0,C 180,E1 -18414.758,E2 -18414.758} C_VEL
LIN {X 0,Y 279.981,Z 608.106,A -85,B 0,C 180,E1 -18415.853,E2 -18415.853} C_VEL
LIN {X 0,Y 277.316,Z 621.659,A -85,B 0,C 180,E1 -18417.2,E2 -18417.2} C_VEL
LIN {X 0,Y 274.312,Z 634.265,A -85,B 0,C 180,E1 -18418.747,E2 -18418.747} C_VEL
LIN {X 0,Y 271.255,Z 645.93,A -85,B 0,C 180,E1 -18420.51,E2 -18420.51} C_VEL
LIN {X 0,Y 267.893,Z 657.625,A -85,B 0,C 180,E1 -18422.671,E2 -18422.671} C_VEL
LIN {X 0,Y 265.487,Z 665.983,A -85,B 0,C 180,E1 -18424.526,E2 -18424.526} C_VEL
LIN {X 0,Y 262.371,Z 675.827,A -85,B 0,C 180,E1 -18427.145,E2 -18427.145} C_VEL
LIN {X 0,Y 259.823,Z 684.002,A -85,B 0,C 180,E1 -18429.826,E2 -18429.826} C_VEL
LIN {X 0,Y 257.7,Z 691.003,A -85,B 0,C 180,E1 -18432.653,E2 -18432.653} C_VEL
LIN {X 0,Y 256.094,Z 697.02,A -85,B 0,C 180,E1 -18435.701,E2 -18435.701} C_VEL
LIN {X 0,Y 254.917,Z 701.847,A -85,B 0,C 180,E1 -18438.873,E2 -18438.873} C_VEL
LIN {X 0,Y 254.242,Z 705.374,A -85,B 0,C 180,E1 -18442.056,E2 -18442.056} C_VEL
LIN {X 0,Y 253.972,Z 707.694,A -85,B 0,C 180,E1 -18445.238,E2 -18445.238} C_VEL
LIN {X 0,Y 253.954,Z 708.858,A -85,B 0,C 180,E1 -18448.414,E2 -18448.414} C_VEL
LIN {X 0,Y 253.955,Z 708.856,A -85,B 0,C 180,E1 -18451.586,E2 -18451.586} C_VEL
LIN {X 0,Y 253.951,Z 707.593,A -85,B 0,C 180,E1 -18454.941,E2 -18454.941} C_VEL
LIN {X 0,Y 254.243,Z 705.349,A -85,B 0,C 180,E1 -18457.945,E2 -18457.945} C_VEL
LIN {X 0,Y 254.919,Z 701.802,A -85,B 0,C 180,E1 -18461.127,E2 -18461.127} C_VEL
LIN {X 0,Y 256.1,Z 696.958,A -85,B 0,C 180,E1 -18464.299,E2 -18464.299} C_VEL
LIN {X 0,Y 257.782,Z 690.69,A -85,B 0,C 180,E1 -18467.452,E2 -18467.452} C_VEL
LIN {X 0,Y 260.175,Z 682.856,A -85,B 0,C 180,E1 -18470.559,E2 -18470.559} C_VEL
LIN {X 0,Y 263.572,Z 676.395,A -85,B 0,C 180,E1 -18473.576,E2 -18473.576} C_VEL
LIN {X 0,Y 267.777,Z 668.529,A -85,B 0,C 180,E1 -18476.499,E2 -18476.499} C_VEL
LIN {X 0,Y 272.871,Z 659.081,A -85,B 0,C 180,E1 -18479.299,E2 -18479.299} C_VEL
LIN {X 0,Y 278.763,Z 647.797,A -85,B 0,C 180,E1 -18481.968,E2 -18481.968} C_VEL
LIN {X 0,Y 284.602,Z 636.151,A -85,B 0,C 180,E1 -18484.18,E2 -18484.18} C_VEL
LIN {X 0,Y 291.1,Z 622.451,A -85,B 0,C 180,E1 -18486.264,E2 -18486.264} C_VEL
LIN {X 0,Y 296.639,Z 609.773,A -85,B 0,C 180,E1 -18487.809,E2 -18487.809} C_VEL
LIN {X 0,Y 302.649,Z 594.699,A -85,B 0,C 180,E1 -18489.256,E2 -18489.256} C_VEL
LIN {X 0,Y 307.994,Z 579.725,A -85,B 0,C 180,E1 -18490.352,E2 -18490.352} C_VEL
LIN {X 0,Y 312.296,Z 565.726,A -85,B 0,C 180,E1 -18491.167,E2 -18491.167} C_VEL
LIN {X 0,Y 316.912,Z 547.466,A -85,B 0,C 180,E1 -18491.972,E2 -18491.972} C_VEL
LIN {X 0,Y 332.323,Z 481.004,A -85,B 0,C 180,E1 -18494.578,E2 -18494.578} C_VEL
LIN {X 0,Y 332.539,Z 480.136,A -85,B 0,C 180,E1 -18494.606,E2 -18494.606} C_VEL
LIN {X 0,Y 332.413,Z 479.678,A -85,B 0,C 180,E1 -18495.099,E2 -18495.099} C_VEL
LIN {X 0,Y 332.212,Z 479.755,A -85,B 0,C 180,E1 -18497.393,E2 -18497.393} C_VEL
LIN {X 0,Y 332.33,Z 480.5,A -85,B 0,C 180,E1 -18498.229,E2 -18498.229} C_VEL
LIN {X 0,Y 314.591,Z 554.223,A -85,B 0,C 180,E1 -18501.382,E2 -18501.382} C_VEL
LIN {X 0,Y 310.69,Z 567.764,A -85,B 0,C 180,E1 -18502.151,E2 -18502.151} C_VEL
LIN {X 0,Y 306.171,Z 581.279,A -85,B 0,C 180,E1 -18503.153,E2 -18503.153} C_VEL
LIN {X 0,Y 300.901,Z 595.213,A -85,B 0,C 180,E1 -18504.48,E2 -18504.48} C_VEL
LIN {X 0,Y 295.887,Z 607.066,A -85,B 0,C 180,E1 -18505.865,E2 -18505.865} C_VEL
LIN {X 0,Y 290.703,Z 618.3,A -85,B 0,C 180,E1 -18507.458,E2 -18507.458} C_VEL
LIN {X 0,Y 284.635,Z 630.401,A -85,B 0,C 180,E1 -18509.591,E2 -18509.591} C_VEL
LIN {X 0,Y 278.485,Z 641.831,A -85,B 0,C 180,E1 -18512.168,E2 -18512.168} C_VEL
LIN {X 0,Y 273.068,Z 651.245,A -85,B 0,C 180,E1 -18514.871,E2 -18514.871} C_VEL
LIN {X 0,Y 268.161,Z 658.899,A -85,B 0,C 180,E1 -18517.665,E2 -18517.665} C_VEL
LIN {X 0,Y 264.184,Z 664.929,A -85,B 0,C 180,E1 -18520.578,E2 -18520.578} C_VEL
LIN {X 0,Y 261.676,Z 668.52,A -85,B 0,C 180,E1 -18522.817,E2 -18522.817} C_VEL
LIN {X 0,Y 259,Z 672.041,A -85,B 0,C 180,E1 -18525.865,E2 -18525.865} C_VEL
LIN {X 0,Y 256.997,Z 674.225,A -85,B 0,C 180,E1 -18528.964,E2 -18528.964} C_VEL
LIN {X 0,Y 255.545,Z 675.097,A -85,B 0,C 180,E1 -18532.096,E2 -18532.096} C_VEL
LIN {X 0,Y 254.697,Z 674.624,A -85,B 0,C 180,E1 -18535.252,E2 -18535.252} C_VEL
LIN {X 0,Y 254.272,Z 672.783,A -85,B 0,C 180,E1 -18538.416,E2 -18538.416} C_VEL
LIN {X 0,Y 254.176,Z 669.508,A -85,B 0,C 180,E1 -18541.585,E2 -18541.585} C_VEL
LIN {X 0,Y 254.203,Z 666.068,A -85,B 0,C 180,E1 -18543.963,E2 -18543.963} C_VEL
LIN {X 0,Y 254.506,Z 660.01,A -85,B 0,C 180,E1 -18547.138,E2 -18547.138} C_VEL
LIN {X 0,Y 254.96,Z 653.172,A -85,B 0,C 180,E1 -18549.921,E2 -18549.921} C_VEL
LIN {X 0,Y 255.615,Z 646.021,A -85,B 0,C 180,E1 -18552.303,E2 -18552.303} C_VEL
LIN {X 0,Y 256.609,Z 637.49,A -85,B 0,C 180,E1 -18554.675,E2 -18554.675} C_VEL
LIN {X 0,Y 257.712,Z 627.246,A -85,B 0,C 180,E1 -18557.047,E2 -18557.047} C_VEL
LIN {X 0,Y 259.186,Z 616.07,A -85,B 0,C 180,E1 -18559.195,E2 -18559.195} C_VEL
LIN {X 0,Y 260.755,Z 602.561,A -85,B 0,C 180,E1 -18561.338,E2 -18561.338} C_VEL
LIN {X 0,Y 262.462,Z 589.205,A -85,B 0,C 180,E1 -18563.055,E2 -18563.055} C_VEL
LIN {X 0,Y 264.03,Z 574.411,A -85,B 0,C 180,E1 -18564.577,E2 -18564.577} C_VEL
LIN {X 0,Y 265.268,Z 560.117,A -85,B 0,C 180,E1 -18565.737,E2 -18565.737} C_VEL
LIN {X 0,Y 266.451,Z 544.385,A -85,B 0,C 180,E1 -18566.694,E2 -18566.694} C_VEL
LIN {X 0,Y 272.585,Z 442.964,A -85,B 0,C 180,E1 -18570.913,E2 -18570.913} C_VEL
LIN {X 0,Y 269.141,Z 418.441,A -85,B 0,C 180,E1 -18572.285,E2 -18572.285} C_VEL
LIN {X 0,Y 262.081,Z 398.428,A -85,B 0,C 180,E1 -18573.832,E2 -18573.832} C_VEL
LIN {X 0,Y 259.466,Z 387.017,A -85,B 0,C 180,E1 -18577.274,E2 -18577.274} C_VEL
LIN {X 0,Y 258.508,Z 383.022,A -85,B 0,C 180,E1 -18578.612,E2 -18578.612} C_VEL
LIN {X 0,Y 258.835,Z 383.175,A -85,B 0,C 180,E1 -18579.057,E2 -18579.057} C_VEL
LIN {X 0,Y 261.201,Z 385.312,A -85,B 0,C 180,E1 -18580.223,E2 -18580.223} C_VEL
LIN {X 0,Y 264.682,Z 393.984,A -85,B 0,C 180,E1 -18583.136,E2 -18583.136} C_VEL
LIN {X 0,Y 265.64,Z 396.145,A -85,B 0,C 180,E1 -18583.724,E2 -18583.724} C_VEL
LIN {X 0,Y 271.762,Z 406.1,A -85,B 0,C 180,E1 -18585.422,E2 -18585.422} C_VEL
LIN {X 0,Y 280.15,Z 421.357,A -85,B 0,C 180,E1 -18587.604,E2 -18587.604} C_VEL
LIN {X 0,Y 287.459,Z 436.803,A -85,B 0,C 180,E1 -18589.415,E2 -18589.415} C_VEL
LIN {X 0,Y 290.224,Z 443.733,A -85,B 0,C 180,E1 -18590.099,E2 -18590.099} C_VEL
LIN {X 0,Y 291.401,Z 453.222,A -85,B 0,C 180,E1 -18590.588,E2 -18590.588} C_VEL
LIN {X 0,Y 286.223,Z 563.329,A -85,B 0,C 180,E1 -18593.236,E2 -18593.236} C_VEL
LIN {X 0,Y 284.756,Z 579.267,A -85,B 0,C 180,E1 -18593.841,E2 -18593.841} C_VEL
LIN {X 0,Y 282.747,Z 594.39,A -85,B 0,C 180,E1 -18594.696,E2 -18594.696} C_VEL
LIN {X 0,Y 280.368,Z 608.578,A -85,B 0,C 180,E1 -18595.786,E2 -18595.786} C_VEL
LIN {X 0,Y 277.805,Z 621.422,A -85,B 0,C 180,E1 -18597.049,E2 -18597.049} C_VEL
LIN {X 0,Y 274.777,Z 634.151,A -85,B 0,C 180,E1 -18598.591,E2 -18598.591} C_VEL
LIN {X 0,Y 271.409,Z 646.986,A -85,B 0,C 180,E1 -18600.528,E2 -18600.528} C_VEL
LIN {X 0,Y 268.025,Z 658.615,A -85,B 0,C 180,E1 -18602.685,E2 -18602.685} C_VEL
LIN {X 0,Y 265.215,Z 668.404,A -85,B 0,C 180,E1 -18604.913,E2 -18604.913} C_VEL
LIN {X 0,Y 262.102,Z 677.975,A -85,B 0,C 180,E1 -18607.536,E2 -18607.536} C_VEL
LIN {X 0,Y 259.599,Z 685.95,A -85,B 0,C 180,E1 -18610.22,E2 -18610.22} C_VEL
LIN {X 0,Y 257.39,Z 693.376,A -85,B 0,C 180,E1 -18613.339,E2 -18613.339} C_VEL
LIN {X 0,Y 255.788,Z 699.269,A -85,B 0,C 180,E1 -18616.494,E2 -18616.494} C_VEL
LIN {X 0,Y 254.941,Z 702.751,A -85,B 0,C 180,E1 -18618.874,E2 -18618.874} C_VEL
LIN {X 0,Y 254.244,Z 706.302,A -85,B 0,C 180,E1 -18622.055,E2 -18622.055} C_VEL
LIN {X 0,Y 253.926,Z 708.644,A -85,B 0,C 180,E1 -18625.237,E2 -18625.237} C_VEL
LIN {X 0,Y 253.942,Z 709.832,A -85,B 0,C 180,E1 -18628.414,E2 -18628.414} C_VEL
LIN {X 0,Y 253.943,Z 709.844,A -85,B 0,C 180,E1 -18631.586,E2 -18631.586} C_VEL
LIN {X 0,Y 253.952,Z 708.612,A -85,B 0,C 180,E1 -18634.941,E2 -18634.941} C_VEL
LIN {X 0,Y 254.244,Z 706.407,A -85,B 0,C 180,E1 -18637.944,E2 -18637.944} C_VEL
LIN {X 0,Y 254.926,Z 702.913,A -85,B 0,C 180,E1 -18641.127,E2 -18641.127} C_VEL
LIN {X 0,Y 256.128,Z 698.129,A -85,B 0,C 180,E1 -18644.297,E2 -18644.297} C_VEL
LIN {X 0,Y 257.805,Z 691.924,A -85,B 0,C 180,E1 -18647.45,E2 -18647.45} C_VEL
LIN {X 0,Y 260.205,Z 684.128,A -85,B 0,C 180,E1 -18650.556,E2 -18650.556} C_VEL
LIN {X 0,Y 262.818,Z 675.816,A -85,B 0,C 180,E1 -18653.23,E2 -18653.23} C_VEL
LIN {X 0,Y 265.605,Z 667.202,A -85,B 0,C 180,E1 -18655.515,E2 -18655.515} C_VEL
LIN {X 0,Y 268.457,Z 657.384,A -85,B 0,C 180,E1 -18657.689,E2 -18657.689} C_VEL
LIN {X 0,Y 271.902,Z 645.516,A -85,B 0,C 180,E1 -18659.839,E2 -18659.839} C_VEL
LIN {X 0,Y 274.989,Z 633.642,A -85,B 0,C 180,E1 -18661.596,E2 -18661.596} C_VEL
LIN {X 0,Y 278.026,Z 620.786,A -85,B 0,C 180,E1 -18663.137,E2 -18663.137} C_VEL
LIN {X 0,Y 280.739,Z 607.252,A -85,B 0,C 180,E1 -18664.439,E2 -18664.439} C_VEL
LIN {X 0,Y 282.956,Z 593.377,A -85,B 0,C 180,E1 -18665.491,E2 -18665.491} C_VEL
LIN {X 0,Y 284.954,Z 578.726,A -85,B 0,C 180,E1 -18666.294,E2 -18666.294} C_VEL
LIN {X 0,Y 286.315,Z 563.827,A -85,B 0,C 180,E1 -18666.859,E2 -18666.859} C_VEL
LIN {X 0,Y 290.777,Z 467.807,A -85,B 0,C 180,E1 -18669.185,E2 -18669.185} C_VEL
LIN {X 0,Y 291.522,Z 451.874,A -85,B 0,C 180,E1 -18669.564,E2 -18669.564} C_VEL
LIN {X 0,Y 289.97,Z 442.572,A -85,B 0,C 180,E1 -18670.111,E2 -18670.111} C_VEL
LIN {X 0,Y 283.635,Z 428.413,A -85,B 0,C 180,E1 -18671.66,E2 -18671.66} C_VEL
LIN {X 0,Y 280.986,Z 424.143,A -85,B 0,C 180,E1 -18672.284,E2 -18672.284} C_VEL
LIN {X 0,Y 275.601,Z 418.382,A -85,B 0,C 180,E1 -18673.507,E2 -18673.507} C_VEL
LIN {X 0,Y 271.061,Z 414.174,A -85,B 0,C 180,E1 -18674.573,E2 -18674.573} C_VEL
LIN {X 0,Y 266.905,Z 409.496,A -85,B 0,C 180,E1 -18675.63,E2 -18675.63} C_VEL
LIN {X 0,Y 258.058,Z 395.193,A -85,B 0,C 180,E1 -18678.288,E2 -18678.288} C_VEL
LIN {X 0,Y 254.17,Z 385.717,A -85,B 0,C 180,E1 -18681.69,E2 -18681.69} C_VEL
LIN {X 0,Y 250.886,Z 378.336,A -85,B 0,C 180,E1 -18684.663,E2 -18684.663} C_VEL
LIN {X 0,Y 249.106,Z 374.528,A -85,B 0,C 180,E1 -18686.38,E2 -18686.38} C_VEL
LIN {X 0,Y 249.015,Z 374.092,A -85,B 0,C 180,E1 -18686.85,E2 -18686.85} C_VEL
LIN {X 0,Y 249.049,Z 374.078,A -85,B 0,C 180,E1 -18691.332,E2 -18691.332} C_VEL
LIN {X 0,Y 249.102,Z 374.08,A -85,B 0,C 180,E1 -18694.963,E2 -18694.963} C_VEL
LIN {X 0,Y 249.089,Z 374.061,A -85,B 0,C 180,E1 -18698.605,E2 -18698.605} C_VEL
LIN {X 0,Y 249.196,Z 374.043,A -85,B 0,C 180,E1 -18703.619,E2 -18703.619} C_VEL
LIN {X 0,Y 249.234,Z 374.036,A -85,B 0,C 180,E1 -18708.616,E2 -18708.616} C_VEL
LIN {X 0,Y 249.447,Z 374.039,A -85,B 0,C 180,E1 -18711.902,E2 -18711.902} C_VEL
LIN {X 0,Y 249.28,Z 374.028,A -85,B 0,C 180,E1 -18715.148,E2 -18715.148} C_VEL
LIN {X 0,Y 249.672,Z 374.01,A -85,B 0,C 180,E1 -18718.387,E2 -18718.387} C_VEL
LIN {X 0,Y 249.674,Z 373.978,A -85,B 0,C 180,E1 -18721.613,E2 -18721.613} C_VEL
LIN {X 0,Y 249.432,Z 374.015,A -85,B 0,C 180,E1 -18726.471,E2 -18726.471} C_VEL
LIN {X 0,Y 249.343,Z 374.036,A -85,B 0,C 180,E1 -18729.736,E2 -18729.736} C_VEL
LIN {X 0,Y 249.178,Z 374.044,A -85,B 0,C 180,E1 -18734.705,E2 -18734.705} C_VEL
LIN {X 0,Y 249.116,Z 374.063,A -85,B 0,C 180,E1 -18738.079,E2 -18738.079} C_VEL
LIN {X 0,Y 249.086,Z 374.073,A -85,B 0,C 180,E1 -18741.518,E2 -18741.518} C_VEL
LIN {X 0,Y 249.131,Z 374.055,A -85,B 0,C 180,E1 -18745.482,E2 -18745.482} C_VEL
LIN {X 0,Y 249.074,Z 374.068,A -85,B 0,C 180,E1 -18748.989,E2 -18748.989} C_VEL
LIN {X 0,Y 249.03,Z 374.091,A -85,B 0,C 180,E1 -18752.426,E2 -18752.426} C_VEL
LIN {X 0,Y 249.039,Z 374.128,A -85,B 0,C 180,E1 -18755.99,E2 -18755.99} C_VEL
LIN {X 0,Y 249.24,Z 374.999,A -85,B 0,C 180,E1 -18756.476,E2 -18756.476} C_VEL
LIN {X 0,Y 250.623,Z 377.654,A -85,B 0,C 180,E1 -18757.406,E2 -18757.406} C_VEL
LIN {X 0,Y 251.611,Z 378.817,A -85,B 0,C 180,E1 -18757.916,E2 -18757.916} C_VEL
LIN {X 0,Y 255.526,Z 386.029,A -85,B 0,C 180,E1 -18760.266,E2 -18760.266} C_VEL
LIN {X 0,Y 259.328,Z 392.807,A -85,B 0,C 180,E1 -18762.284,E2 -18762.284} C_VEL
LIN {X 0,Y 268.869,Z 406.834,A -85,B 0,C 180,E1 -18765.01,E2 -18765.01} C_VEL
LIN {X 0,Y 272.887,Z 415.07,A -85,B 0,C 180,E1 -18766.147,E2 -18766.147} C_VEL
LIN {X 0,Y 280.296,Z 432.217,A -85,B 0,C 180,E1 -18768.172,E2 -18768.172} C_VEL
LIN {X 0,Y 284.91,Z 443.493,A -85,B 0,C 180,E1 -18769.37,E2 -18769.37} C_VEL
LIN {X 0,Y 285.583,Z 450.168,A -85,B 0,C 180,E1 -18769.702,E2 -18769.702} C_VEL
LIN {X 0,Y 280.02,Z 565.027,A -85,B 0,C 180,E1 -18772.51,E2 -18772.51} C_VEL
LIN {X 0,Y 278.523,Z 580.314,A -85,B 0,C 180,E1 -18773.125,E2 -18773.125} C_VEL
LIN {X 0,Y 276.458,Z 595.089,A -85,B 0,C 180,E1 -18773.994,E2 -18773.994} C_VEL
LIN {X 0,Y 273.948,Z 609.094,A -85,B 0,C 180,E1 -18775.101,E2 -18775.101} C_VEL
LIN {X 0,Y 270.985,Z 623.381,A -85,B 0,C 180,E1 -18776.574,E2 -18776.574} C_VEL
LIN {X 0,Y 267.554,Z 636.854,A -85,B 0,C 180,E1 -18778.308,E2 -18778.308} C_VEL
LIN {X 0,Y 264.178,Z 649.135,A -85,B 0,C 180,E1 -18780.298,E2 -18780.298} C_VEL
LIN {X 0,Y 260.504,Z 661.148,A -85,B 0,C 180,E1 -18782.701,E2 -18782.701} C_VEL
LIN {X 0,Y 257.656,Z 670.426,A -85,B 0,C 180,E1 -18784.989,E2 -18784.989} C_VEL
LIN {X 0,Y 254.607,Z 679.519,A -85,B 0,C 180,E1 -18787.695,E2 -18787.695} C_VEL
LIN {X 0,Y 252.129,Z 687.06,A -85,B 0,C 180,E1 -18790.458,E2 -18790.458} C_VEL
LIN {X 0,Y 249.977,Z 694.095,A -85,B 0,C 180,E1 -18793.672,E2 -18793.672} C_VEL
LIN {X 0,Y 248.412,Z 699.619,A -85,B 0,C 180,E1 -18796.919,E2 -18796.919} C_VEL
LIN {X 0,Y 247.508,Z 703.781,A -85,B 0,C 180,E1 -18800.191,E2 -18800.191} C_VEL
LIN {X 0,Y 246.974,Z 706.695,A -85,B 0,C 180,E1 -18803.464,E2 -18803.464} C_VEL
LIN {X 0,Y 246.839,Z 708.432,A -85,B 0,C 180,E1 -18806.736,E2 -18806.736} C_VEL
LIN {X 0,Y 246.857,Z 709.023,A -85,B 0,C 180,E1 -18810,E2 -18810} C_VEL
LIN {X 0,Y 246.84,Z 708.425,A -85,B 0,C 180,E1 -18813.265,E2 -18813.265} C_VEL
LIN {X 0,Y 246.974,Z 706.677,A -85,B 0,C 180,E1 -18816.536,E2 -18816.536} C_VEL
LIN {X 0,Y 247.508,Z 703.746,A -85,B 0,C 180,E1 -18819.81,E2 -18819.81} C_VEL
LIN {X 0,Y 248.417,Z 699.563,A -85,B 0,C 180,E1 -18823.081,E2 -18823.081} C_VEL
LIN {X 0,Y 249.979,Z 694.027,A -85,B 0,C 180,E1 -18826.329,E2 -18826.329} C_VEL
LIN {X 0,Y 252.141,Z 686.986,A -85,B 0,C 180,E1 -18829.541,E2 -18829.541} C_VEL
LIN {X 0,Y 252.796,Z 684.992,A -85,B 0,C 180,E1 -18830.336,E2 -18830.336} C_VEL
LIN {X 0,Y 257.139,Z 677.313,A -85,B 0,C 180,E1 -18834.203,E2 -18834.203} C_VEL
LIN {X 0,Y 261.549,Z 669.826,A -85,B 0,C 180,E1 -18837.181,E2 -18837.181} C_VEL
LIN {X 0,Y 266.899,Z 660.847,A -85,B 0,C 180,E1 -18840.021,E2 -18840.021} C_VEL
LIN {X 0,Y 273.056,Z 650.162,A -85,B 0,C 180,E1 -18842.718,E2 -18842.718} C_VEL
